(**************************************************************************************************************)
(*----------   P1 - ERECTOR   ----------*)
(* All P1 control bits and words must be within address MD3040~MD3079*)
(* All bits and words within the address will be reset when not in autorun mode*)
(**************************************************************************************************************)

	A1_RunStep 				AT %MW3040:INT;

(**************************************************************************************************************)
(*---------- P2 - EXIT ----------*)
(* All P2 control bits and words must be within address MD3080~MD3119*)
(* All bits and words within the address will be reset when not in autorun mode*)
(**************************************************************************************************************)
	A2_RunStep 				AT %MW3080:INT;

(**************************************************************************************************************)
(*---------- P3 - ELEVATOR ----------*)
(* All P3 control bits and words must be within address MD3120~MD3159*)
(* All bits and words within the address will be reset when not in autorun mode*)
(**************************************************************************************************************)

	A3_RunStep 				AT %MW3120		:INT;
	TapeReel_ActivatedL		AT %MX3122.0	:BOOL;
	TapeReel_ActivatedR		AT %MX3122.1	:BOOL;	
	
(**************************************************************************************************************)
(*---------- P4 - HORIZONTAL ----------*)
(* All P4 control bits and words must be within address MD3160~MD3199*)
(* All bits and words within the address will be reset when not in autorun mode*)
(**************************************************************************************************************)

	A4_RunStep 				AT %MW3160 :INT;

(**************************************************************************************************************)
(*---------- P5 SPARE ---------*)
(* All P5 control bits and words must be within address MD3200~MD3239*)
(* All bits and words within the address will be reset when not in autorun mode*)
(**************************************************************************************************************)

	A5_RunStep 				AT %MW3200:INT;

(**************************************************************************************************************)
(*---------- P6 SPARE ----------*)
(* All P6 control bits and words must be within address MD3240~MD3279*)
(* All bits and words within the address will be reset when not in autorun mode*)
(**************************************************************************************************************)

	A6_RunStep  			AT %MW3240 :INT;

(**************************************************************************************************************)
(*---------- P7 SPARE ----------*)
(* All P7 control bits and words must be within address MD3280~MD3319*)
(* All bits and words within the address will be reset when not in autorun mode*)
(**************************************************************************************************************)

	A7_RunStep 				AT %MW3280:INT;

(**************************************************************************************************************)
(*---------- P8 SPARE ----------*)
(* All P8 control bits and words must be within address MD3320~MD3359*)
(* All bits and words within the address will be reset when not in autorun mode*)
(**************************************************************************************************************)

	A8_RunStep 				AT %MW3320:INT;

	
	
	INPUT_TEST		AT %I* 	:INT;
	OUTPUT_TEST		AT %Q* 	:INT;

	I_Reset_HMI: BOOL;
END_VAR

// ---- GVLs/MC/GVL_Holding.TcGVL
VAR_GLOBAL RETAIN PERSISTENT
	
	(* Process Memory*)
	H_CO_StkRdyForXPush					:BOOL;	(*Stack Ready for X Pusher. Do not Stack up if ON*)
	H_CO_StkRdyForYPush					:BOOL;	(*Stack Ready for Y Pusher. Do not activate X Pusher if ON*)
	
	H_ServiceStop_Pressed				:BOOL;	(* Service Stop Pressed *)
	StackerFault_Triggered				:BOOL;
	XPusherFault_Triggered				:BOOL;
	YPusherFault_Triggered				:BOOL;
	ErectorFault_Triggered				:BOOL;
	ExitFault_Triggered					:BOOL;
	HorizontalFault_Triggered			:BOOL;
	MajorFault_Triggered				:BOOL;

		
	H_ER_CtnErected						:BOOL;	(*Carton Erected *)
	H_ER_CtnRdyForPushIn				:BOOL;	(*Carton Erected and Moving Side Flaps Closed. Ready for Stack Push In*)
	H_ER_CtnPushInDone					:BOOL;	(*Stack Pushed into Carton Done, Wait for Side Flap Close. Do not activate Push in if ON*)
	H_ER_CtnSideFlapDone				:BOOL;	(*Carton Side Flap Closing Done. Ready for Glueing*)
	H_ER_CtnRdyForGlue					:BOOL;	(*Carton Pushed into Exit Area Ready for Glueing.*)
	H_ER_CtnGlueDone					:BOOL;	(*Carton Glueing Done. Ready for Exit Send Out*)
	H_ER_CtnWeightOK					:BOOL;	(*Carton Weight Checking OK - At Glueing Area*)

	H_EL_CtnTapeDone					:BOOL;	(*Carton Tape Sealing Done - If ON, send out to exit during origin*)	
	H_EL_CtnWeightOK					:BOOL;	(*Carton Weight Checking OK - On Elevator*)
	H_CartonWeight						:REAL;
	
	H_HOR_CtnTapeDone					:BOOL;	(*Carton Tape Sealing Done - If ON, send out to exit during origin*)	
	H_HOR_CtnWeightOK					:BOOL;	(*Carton Weight Checking OK - On Elevator*)
	
	CaseBufferEmptying_Counter			:INT;
	CaseBufferEmptying_Setting			:INT;
	GlueEmptying_Counter				:INT;
	GlueEmptying_Setting				:INT;
	TapeLow_Setting						:INT;

	
	H_ER_WA_Srv_ZeroOffset				:REAL;	(*Set Zero Point for Case Min C = 180mm	*)
	H_ER_BufCvL_WA_Srv_ZeroOffset		:REAL;	(*Set Zero Point for Case Min B+C = 330mm, where B=2xFlap Width	*)
	H_ER_FlapL_WA_Srv_ZeroOffset		:REAL;	(*Set Zero Point for Case Min A = 200mm	*)
	H_ER_BufCvR_WA_Srv_ZeroOffset		:REAL;	(*Set Zero Point for Case Min B+C = 330mm, where B=2xFlap Width	*)
	H_ER_FlapR_WA_Srv_ZeroOffset		:REAL;	(*Set Zero Point for Case Min A = 200mm	*)
	H_EX_HeightL_WA_Srv_ZeroOffset		:REAL;	(*set Zero Point for Case Min B = 150mm*)
	H_EX_HeightR_WA_Srv_ZeroOffset		:REAL;	(*set Zero Point for Case Min B = 150mm*)
	H_EX_WA_Srv_ZeroOffset				:REAL;	(*Set Zero Point for Case Min C = 180mm*)
	H_CO_CV_WA_Srv_ZeroOffset			:REAL;	
	H_CO_Stopper_WA_Srv_ZeroOffset		:REAL;	
	H_EX_TopL_WA_Srv_ZeroOffset			:REAL;
	H_EX_TopR_WA_Srv_ZeroOffset			:REAL;
	H_CO_FFlapGuide_WA_Srv_ZeroOffset	:REAL;	(*Set Zero Point where Carton min A = 200mm*)

	H_CO_XPush_Srv_EndDatumPos:REAL;		(*Teach End Datum Point at Final Pushing Position for Carton min A = 200mm*)

	H_CO_YPush_Srv_BufFinalPos:REAL;		(*Teach Final Pushing Position to Push Stack onto Buffer Area Before Carton*)
	H_CO_YPush_Srv_CtnFinalPos:REAL;		(*Teach Final Pushing Position to Push Stack into Carton*)	
	H_CO_YPush_Srv_SafePosition:Real;	
	
	H_ER_Arm_Srv_CtnVacuumPos: REAL;		(*Teach Position for Erector cylinder to move up and ready for Vacuum*)
	H_ER_Arm_Srv_CtnErectPos: REAL;			(*Teach Position for Erector Arm to move to final carton erecting position*)

	H_EL_Srv_CtnLoadPos:REAL;				(*Teach Position for Elevator Carton Loading from Tilt Position*)
	H_EL_Srv_CtnRejectExitPos:REAL;			(*Teach Position for Elevator Reject Carton Exit Conveyor Position*)
	H_EL_Srv_CtnGoodExitPos:REAL;			(*Teach Position for Elevator Good Carton Exit Conveyor Position*)
	H_EL_Srv_TapeStartPos:REAL;				(*Teach Position for Elevator Taping Start Position (bottom)*)
	H_EL_Srv_TapeEndPos:REAL;				(*Teach Position for Elevator Taping End Position (Top)*)
 
	H_EL_Push_Srv_HomePos:REAL;				(*Set at Zero Point before Carton is pushed but need to avoid taping unit*)
	H_EL_Push_Srv_ExitfinalPos:REAL;		(*Teach Final Pushing Position to Push Carton onto Exit conveyors*)

	H_EL_Center_Srv_HomePos:REAL;			(*Set at Zero Point before to avoid Carton during tilting*)
	H_EL_Center_Srv_EndDatumPos:REAL;		(*Teach Position for Carton Centering to Tilt Vacuum ON for Carton min B=150mm*)
	H_EL_Center_Srv_MidDatumPos:REAL;		(*Teach Position for Elevator Carton Centering for Taping for Carton min B=150mm*)
	
	
	H_ER_Arm_Srv_HomePos: REAL;			
	H_CO_XPush_Srv_HomePos:REAL;			(*Set at Zero Point out of Bundle Stack Area*)
	H_CO_YPush_Srv_HomePos:REAL;			(*Set at Zero Point out of Bundle Buffer Area*)

	H_CO_XPush_Srv_CurrStandbyPos:REAL;			(* Calculated based on bundle size*)
	H_CO_YPush_Srv_CurrStandbyPos:REAL;			(* Calculated based on bundle size*)
	
	H_ER_WA_Srv_TargetPos				:REAL;
	H_ER_BufCvL_WA_Srv_TargetPos		:REAL;
	H_ER_FlapL_WA_Srv_TargetPos			:REAL;
	H_ER_BufCvR_WA_Srv_TargetPos		:REAL;
	H_ER_FlapR_WA_Srv_TargetPos			:REAL;
	H_EX_HeightL_WA_Srv_TargetPos		:REAL;
	H_EX_HeightR_WA_Srv_TargetPos		:REAL;
	H_EX_WA_Srv_TargetPos				:REAL;
	H_CO_CV_WA_Srv_TargetPos			:REAL;	
	H_CO_Stopper_WA_Srv_TargetPos		:REAL;
	H_EX_TopL_WA_Srv_TargetPos			:REAL;
	H_EX_TopR_WA_Srv_TargetPos			:REAL;
	H_CO_FFlapGuide_WA_Srv_TargetPos	:REAL;
	
	H_ER_ValveOffset					:REAL;	
	H_ER_1St_GlueStartPos				:REAL;
	H_ER_1St_GlueStopPos				:REAL;	
	H_ER_2nd_GlueStartPos				:REAL;
	H_ER_2nd_GlueStopPos				:REAL;		
	ER_GlueHold_Time					:TIME;
	
	
	H_CO_Bdl_StkX_Count:INT;	(*Current Stack X Count*)
	H_CO_Bdl_StkY_Count:INT;	(*Current Stack Y Count*)
	H_CO_Bdl_StkZ_Count:INT;	(*Current Stack Z Count*)

	H_CO_Bdl_StkX_Full:BOOL;	(*Current Stack X Full*)
	H_CO_Bdl_StkY_Full:BOOL;	(*Current Stack Y Full*)
	H_CO_Bdl_StkZ_Full:BOOL;	(*Current Stack Z Full*)
	
	
	
	(***************************** Statistic Value ******************************************)
	Statistic_Total_Runtime				:DINT;
	Statistic_Total_UpTime				:DINT;
	Statistic_Total_DownTime			:DINT;
	Statistic_Total_CaseProduce			:DINT;
	Statistic_Total_Good				:DINT;
	Statistic_Total_NG					:DINT;					
	
	Statistic_Man_Total_Runtime			:DINT;
	Statistic_Man_Total_UpTime			:DINT;
	Statistic_Man_Total_DownTime		:DINT;
	Statistic_Man_Total_CaseProduce		:DINT;
	Statistic_Man_Total_Good			:DINT;
	Statistic_Man_Total_NG				:DINT;
	
	Statistic_Shift_StartTimeH			:ARRAY [0..3] OF UINT;
	Statistic_Shift_StartTimeM			:ARRAY [0..3] OF UINT;
	Statistic_Shift_EndTimeH			:ARRAY [0..3] OF UINT;
	Statistic_Shift_EndTimeM			:ARRAY [0..3] OF UINT;	
	
	Statistic_PreviousShift_Number		:UINT;	
	Statistic_CurShift_Number			:UINT;	
	Statistic_CurShift_StartTime		:STRING;
	Statistic_CurShift_EndTime			:STRING;
	Statistic_CurShift_StartDate		:STRING;
	Statistic_CurShift_CaseProduce		:DINT;
	Statistic_CurShift_Good				:DINT;
	Statistic_CurShift_NG				:DINT;
	Statistic_CurShift_UpTime			:DINT;
	Statistic_CurShift_RunTime			:DINT;
	Statistic_CurShift_DownTime			:DINT;
	
	Statistic_Current					:structStatistic;
	Statistic_History					:structStatistic;
	Statistic_Manual					:structStatistic;
	Statistic_Total						:structStatistic;	
	
	Generate_Report						:BOOL;
	
(**************************************************************************************************************)
(* Exit Case Result *)
(**************************************************************************************************************)	
	Exit_Case_Good	:BOOL;
	Exit_Case_NG	:BOOL;	
END_VAR

// ---- GVLs/MC/GVL_Origin.TcGVL
{attribute 'Tc2GvlVarNames'}
VAR_GLOBAL

(**************************************************************************************************************)
(*----------   P0 - COLLATOR   ----------*)
(* All P0 control bits and words must be within address MD4000~MD4039*)
(* All bits and words within the address will be reset when not in autorun mode*)
(**************************************************************************************************************)

	AO0_RunStep					AT %MW4000:INT;

(**************************************************************************************************************)
(*----------   P1 - ERECTOR   ----------*)
(* All P1 control bits and words must be within address MD4040~MD4079*)
(* All bits and words within the address will be reset when not in autorun mode*)
(**************************************************************************************************************)

	AO1_RunStep 				AT %MW4040:INT;
	
(**************************************************************************************************************)
(*---------- P2 - EXIT ----------*)
(* All P2 control bits and words must be within address MD4080~MD4119*)
(* All bits and words within the address will be reset when not in autorun mode*)
(**************************************************************************************************************)
	AO2_RunStep 			AT %MW4080:INT;

(**************************************************************************************************************)
(*---------- P3 - ELEVATOR ----------*)
(* All P3 control bits and words must be within address MD4120~MD4159*)
(* All bits and words within the address will be reset when not in autorun mode*)
(**************************************************************************************************************)

	AO3_RunStep 			AT %MW4120:INT;

(**************************************************************************************************************)
(*---------- P4 HORIZONTAL----------*)
(* All P4 control bits and words must be within address MD4160~MD4199*)
(* All bits and words within the address will be reset when not in autorun mode*)
(**************************************************************************************************************)

	AO4_RunStep 			AT %MW4160 :INT;

(**************************************************************************************************************)
(*---------- P5 SPARE----------*)
(* All P5 control bits and words must be within address MD4200~MD4239*)
(* All bits and words within the address will be reset when not in autorun mode*)
(**************************************************************************************************************)

	AO5_RunStep 			AT %MW4200:INT;

(**************************************************************************************************************)
(*---------- P6 SPARE----------*)
(* All P6 control bits and words must be within address MD4240~MD4279*)
(* All bits and words within the address will be reset when not in autorun mode*)
(**************************************************************************************************************)

	AO6_RunStep  			AT %MW4240 :INT;

(**************************************************************************************************************)
(*---------- P7 SPARE----------*)
(* All P7 control bits and words must be within address MD4280~MD4319*)
(* All bits and words within the address will be reset when not in autorun mode*)
(**************************************************************************************************************)

	AO7_RunStep 			AT %MW4280:INT;

(**************************************************************************************************************)
(*---------- P8 SPARE ----------*)
(* All P8 control bits and words must be within address MD4320~MD4359*)
(* All bits and words within the address will be reset when not in autorun mode*)
(**************************************************************************************************************)

	AO8_RunStep 			AT %MW4320:INT;

	

END_VAR

// ---- GVLs/MC/GVL_Error.TcGVL
{attribute 'Tc2GvlVarNames'}
VAR_GLOBAL
	
(**************************************************************************************************************)
(* warning Flag *)
(**************************************************************************************************************)
W_ER_BufRefill		AT %MX2000.0:BOOL;
W_EX_TapeLRefill	AT %MX2000.1:BOOL;
W_EX_TapeRRefill	AT %MX2000.2:BOOL;
W_CO_IncomingEmpty	AT %MX2000.3:BOOL;
W_HOR_TapeLRefill	AT %MX2001.1:BOOL;
W_HOR_TapeRRefill	AT %MX2001.2:BOOL;
W_HOR_Conv_Full		AT %MX2001.3:BOOL;
W_Glue_Low_Level	AT %MX2001.4:BOOL;
W_Glue_is_Empty		AT %MX2001.5:BOOL;
W_CaseBuffer_is_Empty	AT %MX2001.6:BOOL;
W_ServiceStop		AT %MX2001.7:BOOL;
W_Hor_TapeLowL		AT %MX2002.0:BOOL;
W_Hor_TapeLowR		AT %MX2002.1:BOOL;

(**************************************************************************************************************)
(*General  Error Flag *)
(**************************************************************************************************************)

E_AutorunDataNG :STRING;
E_Erector_FrontDoor_Opn		:BOOL;
E_Erector_RearDoor_Opn		:BOOL;
E_Collator_FrontDoor_Opn	:BOOL;
E_Collator_RearDoor_Opn		:BOOL;
E_Elevator_LeftTopDoor_Opn	:BOOL;
E_Elevator_LeftBtmDoor_Opn	:BOOL;
E_Elevator_RightDoor_Opn	:BOOL;
E_Horizontal_LeftDoor_Opn	:BOOL;
E_Horizontal_RightDoor_Opn	:BOOL;
E_Door_SafetyBroken			:BOOL;
E_Estop_Panel				:BOOL;
E_Estop_Collator			:BOOL;
E_Estop_HorLeft				:BOOL;
E_Estop_HorRight			:BOOL;
E_Estop_HorExit				:BOOL;
E_EStop_SafetyBroken		:BOOL;
E_X_Axis_BundleStackCount	:BOOL;
E_Y_Axis_BundleStackCount	:BOOL;
E_Z_Axis_BundleStackCount	:BOOL;
E_Recipe_H_OutOfTolerance	:BOOL;
E_Recipe_L_OutOfTolerance	:BOOL;
E_Recipe_W_OutOfTolerance	:BOOL;
E_Recipe_A_OutOfTolerance	:BOOL;
E_Recipe_B_OutOfTolerance	:BOOL;
E_Recipe_C_OutOfTolerance	:BOOL;
E_Recipe_A_SmallerThan_W	:BOOL;
E_Recipe_C_SmallerThan_L	:BOOL;
E_Recipe_B_SmallerThan_H	:BOOL;
	
(**************************************************************************************************************)
(*P0  Error Flag *)
(* All P0 control bits and words must be within address MD1000~MD1039*)
(* All bits and words within the address will be reset when error reset*)
(**************************************************************************************************************)
	
	E_Stack_Overflow 						:BOOL;
	E_Stack_Full			AT %MX1000.1	:BOOL;
	E_Door_Open				AT %MX1000.2	:BOOL;
	E_Bundle_Stuck_on_Infeed AT %MX1000.3	:BOOL;
	E_Bundle_Full			AT %MX1000.4	:BOOL;
	E_CAM_Up_Timeout		AT %MX1000.5	:BOOL;
	E_BundleJam_AfterStack	AT %MX1000.6	:BOOL;
	E_BundleJam_atRelease	AT %MX1000.7	:BOOL;	
	E_CAM_Down_Timeout		AT %MX1001.0	:BOOL;
	E_Stack_Full_ON			AT %MX1001.1	:BOOL;
	E_BundleDetected		AT %MX1001.2	:BOOL;
	E_Bundle_Stack_Sensor	AT %MX1001.3	:BOOL;
	E_BundleDetect_Sensor1	AT %MX1002.0	:BOOL;
	E_BundleDetect_Sensor2	AT %MX1002.1	:BOOL;
	E_BundleDetect_Sensor3	AT %MX1002.2	:BOOL;
	E_BundleDetect_Sensor4	AT %MX1002.3	:BOOL;
	E_BundleDetect_Sensor5	AT %MX1002.4	:BOOL;
	E_BundleDetect_Sensor6	AT %MX1002.5	:BOOL;
	E_BundleDetect_Sensor7	AT %MX1002.6	:BOOL;
	E_BundleDetect_Sensor8	AT %MX1002.7	:BOOL;
	
	
(**************************************************************************************************************)
(*P1  Error Flag *)
(* All P1 control bits and words must be within address MD1040~MD1079*)
(* All bits and words within the address will be reset when error reset*)
(**************************************************************************************************************)

	E_Buff1_BundleNotDetect	AT %MX1040.0	:BOOL;
	E_BundleJam_atStaker	AT %MX1040.1	:BOOL;


(**************************************************************************************************************)
(*P2  Error Flag *)
(* All P2 control bits and words must be within address MD1080~MD1119*)
(* All bits and words within the address will be reset when error reset*)
(**************************************************************************************************************)

	E_Buf1_BundleMissing	AT %MX1080.0	:BOOL;	
	E_Buf1_BundleJam		AT %MX1080.1	:BOOL;
	E_GapSensor				AT %MX1080.2	:BOOL;
	E_BundleDetectedinBuf1	AT %MX1080.3	:BOOL;
	E_BundleDetectedinBuf2	AT %MX1080.4	:BOOL;
	E_GapSensorError		AT %MX1080.5	:BOOL;
	E_PTC_BundleNOK			AT %MX1080.6	:BOOL;
	E_Buf1_Sensor			AT %MX1080.7	:BOOL;
	E_Buf2_Sensor			AT %MX1081.0	:BOOL;
	
(**************************************************************************************************************)
(*P3  Error Flag *)
(* All P3 control bits and words must be within addres MD1120~MD1159*)
(* All bits and words within the address will be reset when error reset*)
(**************************************************************************************************************)

	E_NoGapAtStoper				AT %MX1120.0	:BOOL;	
	E_LeftStopper_NotDetect		AT %MX1120.1	:BOOL;	
	E_RightStopper_NotDetect 	AT %MX1120.2	:BOOL;		
	E_ER_BufRefill				AT %MX1120.3	:BOOL;
	E_CaseDetected				AT %MX1120.4	:BOOL;
	E_CaseNotDetected			AT %MX1120.5	:BOOL;
	E_CaseVacuumNotDetected		AT %MX1120.6	:BOOL;
	E_Nordson_Alarm				AT %MX1120.7	:BOOL;
	E_EmptyCaseDetected			AT %MX1121.0	:BOOL;
	E_CaseBufferAlignment_Err	AT %MX1121.1	:BOOL;
	E_CaseBuffer_Not_Ready		AT %MX1121.2	:BOOL;
	E_CaseBuffer_EmptySensors	AT %MX1121.3	:BOOL;
	E_Case_Infeed_Safety_NOk	AT %MX1121.4	:BOOL;
	E_ER_EmptyL_PE				AT %MX1121.5	:BOOL;
	E_ER_BufferL_PE				AT %MX1121.6	:BOOL;
	E_ER_EmptyR_PE				AT %MX1121.7	:BOOL;
	E_ER_BufferR_PE				AT %MX1122.0	:BOOL;
	
(**************************************************************************************************************)
(*P4  Error Flag *)
(* All P4 control bits and words must be within address MD1160~MD1199*)
(* All bits and words within the address will be reset when error reset*)
(**************************************************************************************************************)
	E_WT_Conv_Jam				AT %MX1160.0	:BOOL;	
	E_CartonMissing				AT %MX1160.1	:BOOL;
	E_EX_CartonDetected			AT %MX1160.2	:BOOL;

(**************************************************************************************************************)
(*P5  Error Flag *)
(* All P5 control bits and words must be within address MD1200~MD1239*)
(* All bits and words within the address will be reset when error reset*)
(**************************************************************************************************************)
	E_BeltTension_Right_NOK		AT %MX1200.0	:BOOL;
	E_BeltTension_Left_NOK		AT %MX1200.1	:BOOL;
	E_DriveBeltTension_NOK		AT %MX1200.2	:BOOL;
	E_Weight_CV_CartonNotDetect AT %MX1200.3	:BOOL;
	E_Weight_CV_CartonDetect	AT %MX1200.4	:BOOL;
	E_EL_CartonNotDetect		AT %MX1200.5	:BOOL;
	E_Weigh_ReadingErr			AT %MX1200.6	:BOOL;
	E_Weigh_ConsecutiveErr		AT %MX1200.7	:BOOL;

	E_CartonTapingErrL							:BOOL;
	E_CartonTapingErrR							:BOOL;
(**************************************************************************************************************)
(*P6  Error Flag *)
(* All P6 control bits and words must be within address MD1240~MD1279*)
(* All bits and words within the address will be reset when error reset*)
(**************************************************************************************************************)
	E_Top_Conv_Jam				AT %MX1240.0	:BOOL;
	E_Bottom_Conv_Jam			AT %MX1240.1	:BOOL;
	E_Hor_Entry_Sensor			AT %MX1240.2	:BOOL;
	E_Hor_Exit_Sensor			AT %MX1240.3	:BOOL;
	
(**************************************************************************************************************)
(*P7  Error Flag *)
(* All P7 control bits and words must be within address MD1280~MD1319*)
(* All bits and words within the address will be reset when error reset*)
(**************************************************************************************************************)

(**************************************************************************************************************)
(*P8  Error Flag *)
(* All P8 control bits and words must be within address MD1320~MD1359*)
(* All bits and words within the address will be reset when error reset*)
(**************************************************************************************************************)


END_VAR

// ---- GVLs/MC/GVL_Configuration.TcGVL
VAR_GLOBAL  RETAIN PERSISTENT
	A_Srv_XPusherHiSpeed	:REAL;
	A_Srv_XPusherLoSpeed	:REAL;
	A_Srv_YPusherHiSpeed	:REAL;
	A_Srv_YPusherLoSpeed	:REAL;	

	A_Srv_ErectorArmHiSpeed:REAL;
	A_Srv_ErectorArmLoSpeed:REAL;
	
	A_Srv_ElevAutoHiSpeed:REAL;
	A_Srv_ElevAutoLoSpeed:REAL;
	A_Srv_ElevAutoMidSpeed:REAL:=60000;
	
	
	A_Srv_BeltOriginSpeed:REAL:=10000;
	A_Srv_ElevOriginSpeed:REAL:=1000;
	A_Srv_WAOriginSpeed:REAL:=1000;
	
	A_Srv_BeltAutoHiSpeed:REAL:=50000;	(*200000*)
	A_Srv_BeltAutoLoSpeed:REAL:=30000;	

	A_Srv_Default_Acc:REAL:=1000;
	A_Srv_Default_Dec:REAL:=1000;

	(* 	1 = Operator
		2 = Maintenance
		3 = Supervisor
		4 = Flexlink 
	*)

	Cfg_UserLvl_Operation	:INT	:=1;		
	Cfg_UserLvl_Manual		:INT	:=2;
	Cfg_UserLvl_Recipe		:INT	:=3;
	Cfg_UserLvl_Setting		:INT	:=3;
	Cfg_UserLvl_Config		:INT	:=4;
	

	Cfg_EnbAutoWA			:BOOL	:=TRUE;		(*1=Enable Auto Width Adjust*)
	Cfg_VerticalExit		:BOOL	:=FALSE;	(*1=Enable Vertical Exit with elevator*)
	Cfg_CollDircLtoR		:BOOL	:=FALSE;		(*1=Collator Push In Direction from Left to Right, 0 = Right to Left*)
	Cfg_EnbNordson			:BOOL	:=FALSE;	(*1=Enable Nordson Glueing*)
	Cfg_EnbWeightCheck		:BOOL	:=TRUE;		(*1=Enable Weight Checking*)
	Cfg_HorizontalExit		:BOOL	:=TRUE;		(*1=Enable Horizontal Exit*)
	Cfg_Exit90DegConv		:BOOL	:= FALSE;	(* 1=Enable Exit 90 Deg Conveyor	*)
	Cfg_Upstream_Conveyor	:BOOL	:= TRUE;	(* Upstream conveyor is connected	*)
	Cfg_prodSpeed_perHour	:INT	:= 120;		(* Number of carton produce per minute *)
	
	
	Cfg_BypassCollator:BOOL	:= FALSE;	(*1=Bypass Collator to run Erector and Elevator only*)
	Cfg_BypassErector:BOOL	:= FALSE;	(*1=Bypass Erector to run Collator only*)
	Cfg_BypassHorizontal:BOOL:= FALSE;	(*1=Bypass Horizontal to run Collator only*)
	
	Cfg_CaseA_Min	:REAL	:= 200;	
	Cfg_CaseB_Min	:REAL	:= 150;	
	Cfg_CaseC_Min	:REAL	:= 180;	
	Cfg_BundleW_Min	:REAL	:= 20;	
	Cfg_BundleL_Min	:REAL	:= 70;	
	Cfg_BundleH_Min	:REAL	:= 15;

	Cfg_CaseA_Max	:REAL	:= 640;	
	Cfg_CaseB_Max	:REAL	:= 500;
	Cfg_CaseC_Max	:REAL	:= 640;	
	Cfg_BundleW_Max	:REAL	:= 300;	
	Cfg_BundleL_Max	:REAL	:= 320;	
	Cfg_BundleH_Max	:REAL	:= 150;	
	
END_VAR

// ---- GVLs/MC/GVL_HMI.TcGVL
VAR_GLOBAL
	
	NewRecipe:structRecipe;
	
	
	T_GlobalAckAlarm:BOOL;
	
	T_SimPushIn:BOOL;
	
	T_DisplayWordSelect:WORD;
	T_MonitorWord:WORD;
	T_MonitorByte1Name:STRING;
	T_MonitorByte2Name:STRING;
	T_Monitor2Bytes:BOOL;
	MC_WA_Run	:BOOL;
END_VAR

VAR_GLOBAL RETAIN PERSISTENT

	CurrRecipe		:structRecipe;
	McData			:structMachineData;
	HMI				:structHMI;
	T_GlueEnable	:BOOL;
	T_ExitCvFull	:BOOL;
	
END_VAR

// ---- GVLs/MC/GVL_Status.TcGVL
VAR_GLOBAL
	
END_VAR

// ---- GVLs/MC/GVL_Symbol_Spec.TcGVL
VAR_GLOBAL
	
(*FlexLink Standard Symbol Naming Convention*)
(*
ER = Erector
CO = Collator
EX = Exit
EL = Elevator
WT = Weight checker
PB = push button
PL = push button light
Emg = Emergency Stop
SC = Safety Circuit
Cyl = Cylinder
Srv = Servo Motor
Mtr = AC Motor
Nord = Nordson Dispenser
Alm = Alarm
Rdy = Ready
SFlapL = Side Flap Left
SFlapR = Side Flap Right
BFlapL = Bottom Flap Left
BFlapR = Bottom Flap Right
Stp = Stopper
Ctn = Carton
LC = Light Curtain
Bdl = Bundle
Stk = Stack
Push = Pusher
Brdg = Bridge
Fx = Fixed
Mv = Moving

SC[0] = COLLATOR STACKING
SC[1] = COLLATOR X PUSHER
SC[2] = COLLATOR Y PUSHER & BRIDGE
SC[3] = ERECTOR ARM & SIDE FLAP CLOSE
SC[4] = HOT GLUE & WEIGHT CHECKING 
SC[5] = TILT & ELEVATOR
SC[6] = HORIZONTAL

*)

END_VAR

// ---- GVLs/MC/GVL_Timer.TcGVL
VAR_GLOBAL
	
	CO_Stk_Up_TON: Ton;
	CO_Stk_Dn_TON: Ton;
	CO_Bdl_Count_TON: Ton;
	CO_Bdl_Reach_TON: Ton;
	CO_Bdl_Stack_TON: Ton;
	CO_Bdl_Count_TOFF: Ton;
	CO_Stk_AtBuf_TON: Ton;

	ER_BufCv_Ctn_TON:ton;
	ER_BufCvL_Ctn_TON:ton;
	ER_BufCvR_Ctn_TON:ton;

	TP_Cyl_Timeout: TIME := T#5S;
	
	EL_Ctn_TON: Ton;
	EL_Ctn_TOFF: Ton;
	EL_TopCv_Ctn_TON: Ton;
	EL_TopCv_Ctn_TOFF: Ton;
	EL_BotCv_Ctn_TON: Ton;
	EL_BotCv_Ctn_TOFF: Ton;
	
	CO_Bdl_ZFull_TON: Ton;
	CO_Bdl_XFull_TON: Ton;
	CO_Bdl_ZFull_TOFF: Ton;
	
	pls_CoStkMtrStop: R_trig;
	tmr_CoStkMtrStop: Ton;

	EL_LC_Safety_TON: Ton;
	
	HOR_Ctn_TON: Ton;
	HOR_Ctn_TOFF: Ton;
	HOR_DnStream_TOFF: Ton;
	HOR_TopCv_Ctn_TON: Ton;
	HOR_TopCv_Ctn_TOFF: Ton;
	HOR_BotCv_Ctn_TON: Ton;
	HOR_BotCv_Ctn_TOFF: Ton;
	
	HOR_LC_Safety_TON: Ton;
END_VAR

// ---- POUs/MC/MAIN.TcPOU
PROGRAM MAIN
VAR
	Reset: BOOL;
	MachineEmpty: BOOL;
	plsMemoryReset: R_trig;
	tmrStartWrite: Ton;
	tmrWriteInterval: Ton;
	WritePersistentDataBusy: BOOL;
	plsStartWrite: R_trig;
	InstWritePersistentData:WritePersistentData;
	Timeout:ton;
	Test: BOOL;
	TIMEr: TIME;
	plsPurgeErectorCaseOff	: 	R_trig;
	plsServiceStop			:	R_trig;
	plsMAchineStart			:	R_trig;
	WA_ResetDly:TON;
	MC_Empty:BOOL;
	GetUPSStatus:FB_GetUPSStatus;
	GetFB_LocalSystemTime:FB_LocalSystemTime;
END_VAR


(**************************************************************************************************************)
(* Machine Control *)
(**************************************************************************************************************)

HMI.V_MachineSpeed	:= 100;

Check_AutorunCond();

Check_Ethercat();

MC_Ctrl(
	In_Start_PB					:= I_Start_PB AND NOT W_ServiceStop AND ER_origin.ER_WA_Origin  ,
	In_Stop_PB					:= I_Stop_PB ,
	In_EmgOK					:= I_Emg_SC_OK AND NOT  E_EStop_SafetyBroken,
	In_Door_Sw					:= TRUE(*I_Door_SC_OK AND NOT E_Door_SafetyBroken*),
	In_Pressure_Sw				:= (I_PressSw_OK AND NOT I_Pneumatic_Sup1_ON AND NOT I_Pneumatic_Sup2_ON) OR NOT (I_Door_SC_OK AND Guard_door.Guard_Door_Fault) ,
	In_LightCurtainSafeToCross	:= TRUE(*HOR_LC_Muting*) ,
	In_LightCurtainOK			:= I_HLC_SC_OK  OR NOT I_Door_SC_OK OR Guard_door.Guard_Door_Fault,
	In_CommunicationOK			:= S_ECat_NOK,
	In_IncomingPowerPhase_OK	:= I_IncomingPowerPhase_OK,
	In_OtherTrouble				:= Guard_door.Guard_Door_Fault ,
	In_Reset_PB					:= I_Reset_PB OR I_Reset_HMI ,
	In_Start_Enable				:= A_AutorunDataOK ,
	In_EndProdWPCleared			:= ,
	In_WaitingForMaterial		:= NOT(I_Nord_Rdy OR NOT T_GlueEnable OR mc.DryRun) OR W_Glue_is_Empty	OR W_CaseBuffer_is_Empty,	
	Out_RedTower				=> O_Red_TL ,
	Out_YelTower				=> O_Yel_TL ,
	Out_GrnTower				=> O_Grn_TL ,
	Out_Buzzer					=> O_Buz_TL, 
	Out_StartPL					=> O_Start_PL,
	Out_StopPL					=> O_Stop_PL,
	Out_ResetPL					=> O_Reset_PL,
	McVar 						:= MC,	
	HMI 						:= HMI);


// ************************************************
// Service Stop Memory
IF I_Stop_PB AND mc.autorunning THEN 
	H_ServiceStop_Pressed	:= TRUE;
END_IF

plsMAchineStart	(CLK:= mc.AutoRunning);
IF plsMAchineStart.Q	THEN
	H_ServiceStop_Pressed	:= FALSE;
	MajorFault_Triggered 	:= FALSE;
	StackerFault_Triggered 	:= FALSE;
	XPusherFault_Triggered 	:= FALSE;
	YPusherFault_Triggered 	:= FALSE;
	ErectorFault_Triggered	:= FALSE;
	ExitFault_Triggered		:= FALSE;
	HorizontalFault_Triggered:= FALSE;
END_IF

// *************************************************	
// Service Stop Warning
plsServiceStop (CLK := H_ServiceStop_Pressed AND NOT mc.AutoRunning );
IF plsServiceStop.Q THEN
	W_ServiceStop	:= TRUE;	
END_IF	



// Machine Empty	
MachineEmpty := NOT I_ER_StpL_Ctn_PE AND
				NOT I_ER_StpR_Ctn_PE AND
				NOT I_EX_Cv_Ctn_PE AND
				NOT I_HOR_Entry_Cv_Present AND
				MC.AllStationRdy;

				
O_DoorLock	:= 	(* MC.ManualMode AND 
				I_Pneumatic_Sup1_ON AND 
				I_Pneumatic_Sup2_ON AND*)
				NOT (	mc.AutoRunning OR 
						SC[0].OriginSchRun OR
						SC[1].OriginSchRun OR
						SC[2].OriginSchRun OR
						SC[3].OriginSchRun OR
						SC[4].OriginSchRun OR
						SC[5].OriginSchRun OR
						SC[6].OriginSchRun);				

				
IF 	HMI.T_EndProd AND 
	sc[0].Rdy AND
	sc[1].Rdy AND
	sc[2].Rdy AND
	sc[3].Rdy AND
	sc[4].Rdy AND
	sc[6].Rdy AND	
	MachineEmpty AND
 	mc.AutoRunning THEN
	MC.StopPressed	:= TRUE;
END_IF


IF NOT mc.AutoRunning THEN
	HMI.T_EndProd := FALSE;
END_IF

(**************************************************************************************************************)
(* Calling of Programs *)
(**************************************************************************************************************)
WarningMsg();
Calc_McPerformance();
Std_System_Out();
TouchScreen();
Statistic();
Recipe_Handling();
Guard_Door();
Emergency_Stop();
CO_Main();			(*COLLATOR MAIN PROGRAM*)
ER_Main();			(*ERECTOR MAIN PROGRAM*)
EX_Main();			(*EXIT MAIN PROGRAM*)
(*EL_Main();		(*ELEVATOR MAIN PROGRAM*)*)
HMI.T_Station_BypassP[5] := TRUE;
HOR_Main();			(*HORIZONTAL MAIN PROGRAM*)
Track_and_Trace(); 	(* TRACK AND TRACE PROGRAM *)


(* MACHINE CONDITION *)
MC_Empty	:= NOT( 	I_CO_YStk_AtBuf1_PE OR 
						I_CO_YStk_AtBuf2_PE OR
						I_CO_Bdl_Stack_PE OR
						I_CO_Bdl_PE1 OR
						I_CO_Bdl_PE2 OR
						I_CO_Bdl_PE3 OR
						I_CO_Bdl_PE4 OR
						I_CO_Bdl_PE5 OR
						I_CO_Bdl_ZLimit_PE OR
						I_CO_Bdl_ZFull_PE OR
						I_ER_RefillL_PE OR
						I_ER_BufferL_PE OR
						I_ER_BufferR_PE OR
						I_ER_StpL_Ctn_PE OR
						I_ER_StpR_Ctn_PE OR
						I_EX_Cv_Ctn_PE OR
						I_HOR_Entry_Cv_Present									
												);


IF NOT MC.AutoMode THEN
	Memory_Handling();
END_IF

WA_ResetDly	(IN := NOT (sc[0].OriginSchRun OR
		sc[1].OriginSchRun OR
	 	sc[2].OriginSchRun OR 
		sc[3].OriginSchRun OR
		sc[4].OriginSchRun OR 
		sc[6].OriginSchRun OR	
		HMI.T_OriginSearch OR
		MC.OriginSchRun) AND 
		MC.AllOrigin AND
		MC_WA_Run , pt := T#1S);

		
IF WA_ResetDly.Q THEN
	MC_WA_Run	:=FALSE;
END_IF			

(**************************************************************************************************************)
(* UPS Battery Status *)
(**************************************************************************************************************)
GetUPSStatus(
	sNetId:= '10.1.33.138.1.1' , 
	nPort:= 801, 
	bEnable:=TRUE , 
	bValid=> , 
	bError=> , 
	nErrId=> , 
	stStatus=> );

END_PROGRAM

// ---- POUs/MC/Check_AutorunCond.TcPOU
PROGRAM Check_AutorunCond
VAR
END_VAR


E_AutorunDataNG := '';

	
IF (CurrRecipe.rCaseA < Cfg_CaseA_Min) OR 
	(CurrRecipe.rCaseA > Cfg_CaseA_Max) THEN
	E_AutorunDataNG := 'Case Dimension A out of tolerance';
	E_Recipe_A_OutOfTolerance	:= TRUE;
ELSE
	E_Recipe_A_OutOfTolerance	:= FALSE;
END_IF
	
IF (CurrRecipe.rCaseB < Cfg_CaseB_Min) OR 
	(CurrRecipe.rCaseB > Cfg_CaseB_Max) THEN
	E_AutorunDataNG := 'Case Dimension B out of tolerance';
	E_Recipe_B_OutOfTolerance	:= TRUE;
ELSE
	E_Recipe_B_OutOfTolerance	:= FALSE;
END_IF
	
IF (CurrRecipe.rCaseC < Cfg_CaseC_Min) OR 
	(CurrRecipe.rCaseC > Cfg_CaseC_Max) THEN
	E_AutorunDataNG := 'Case Dimension C out of tolerance';
	E_Recipe_C_OutOfTolerance	:= TRUE;
ELSE
	E_Recipe_C_OutOfTolerance	:= FALSE;
END_IF
		

IF 	E_Recipe_A_OutOfTolerance	OR
	E_Recipe_B_OutOfTolerance	OR
	E_Recipe_C_OutOfTolerance	
THEN	
	A_AutorunDataOK := FALSE;
ELSE
	A_AutorunDataOK := TRUE;	
END_IF

END_PROGRAM

// ---- POUs/MC/Check_Ethercat.TcPOU
PROGRAM Check_Ethercat
VAR
END_VAR


S_ECat_NOK := FALSE;


IF NOT ER.Bypass THEN
	S_ECat_NOK := 	 S_ECat_NOK 
					 OR (I_ECat_41BC1<>8)
					 OR (I_ECat_41DI1<>8)
					 OR (I_ECat_41DI2<>8)
					 OR (I_ECat_41DO1<>8)
					 OR (I_ECat_41DO2<>8)
					(* OR (I_ECat_41CO1<>8)	*)
					 OR (I_ECat_41BC2<>8)
					 OR (I_ECat_41BC3<>8)
					 OR (I_ECat_70A1<>8)
					 OR (I_ECat_71A1<>8)
					 OR (I_ECat_60A1<>8)
					 OR (I_ECat_61A1<>8)
					 OR (I_ECat_62A1<>8)
					 OR (I_ECat_63A1<>8)
					 OR (I_ECat_64A1<>8)
					 OR (I_ECat_65A1<>8)
					 OR (I_ECat_66A1<>8);
END_IF


IF NOT CO.Bypass THEN
	S_ECat_NOK := 		S_ECat_NOK 
					OR (I_ECat_141BC1<>8)
					OR (I_ECat_141DI1<>8)
					OR (I_ECat_141DO1<>8)
					OR (I_ECat_141BC2<>8)
					OR (I_ECat_170A1<>8) 
					OR (I_ECat_160A1<>8)
					OR (I_ECat_161A1<>8)
					OR (I_ECat_162A1<>8)
					OR (I_ECat_162A1<>8);
END_IF



IF NOT HOR.Bypass THEN
	S_ECat_NOK := S_ECat_NOK (*
					OR (I_ECat_241BC1<>8)
					OR (I_ECat_241DI1<>8)
					OR (I_ECat_241DO1<>8)*)
					OR (I_ECat_260A1<>8);
END_IF

END_PROGRAM

// ---- POUs/Erector/ER_Origin.TcPOU
PROGRAM ER_Origin
VAR_IN_OUT
	Station		:structStationCtrl;
END_VAR
VAR
	pls_OriginSchRun: R_trig;
	ER_CtnPresent_Origin:BOOL;
	ER_NoCtnPresent_Origin:BOOL;
	
	ER_WA_Origin: BOOL;
	ER_CtnDone_Origin: BOOL;
	ER_Ctn_OriginState: BOOL;
	TimeoutTrigger: BOOL;
	TimeoutSetting: TIME;
	Timeout:ton;
END_VAR

(**************************************************************************************************************)
(* Station Width Adjust in Origin Condition *)
(**************************************************************************************************************)
ER_WA_Origin := fcCompareWAPos(CurrPos:= ER_WA_Srv_Var.Out_CurrPos, TargetPos:= H_ER_WA_Srv_TargetPos) ;

(**************************************************************************************************************)
(* Station Origin Condition *)
(**************************************************************************************************************)

IF Cfg_CollDircLtoR THEN
	ER_CtnPresent_Origin := (	ER_StpR_Cyl_Var.S_WorkPos AND 
								ER_StpL_Cyl_Var.S_WorkPos AND
								ER_FFlapL_Cyl_Var.S_HomePos AND 
								(*ER_RFlapL_Cyl_Var.S_HomePos AND*)
								ER_FFlapR_Cyl_Var.S_HomePos AND 
								(*ER_RFlapR_Cyl_Var.S_WorkPos AND*)
								ER_TFlapClsL_Cyl_Var.S_WorkPos AND
								ER_TFlapClsR_Cyl_Var.S_WorkPos AND
							(*	ER_BFlapL_Vac_Var.S_Vacuum AND 
								ER_BFlapR_Vac_Var.S_Vacuum AND*)
								I_ER_StpL_Ctn_PE AND I_ER_StpR_Ctn_PE) 
								OR MC.DryRun ;
ELSE
	ER_CtnPresent_Origin := (	ER_StpR_Cyl_Var.S_WorkPos AND 
								ER_StpL_Cyl_Var.S_WorkPos AND
								ER_FFlapL_Cyl_Var.S_WorkPos AND 
								ER_RFlapL_Cyl_Var.S_WorkPos AND
								ER_FFlapR_Cyl_Var.S_HomePos AND 
								ER_RFlapR_Cyl_Var.S_HomePos AND
								(*
								ER_BFlapL_Vac_Var.S_Vacuum AND 
								ER_BFlapR_Vac_Var.S_Vacuum AND*)
								ER_BFlapCloseL_Cyl_Var.S_HomePos AND 
								ER_BFlapCloseR_Cyl_Var.S_HomePos AND
								I_ER_StpL_Ctn_PE AND I_ER_StpR_Ctn_PE)
								OR MC.DryRun ;
END_IF

ER_CtnDone_Origin := (	ER_StpR_Cyl_Var.S_WorkPos AND 
						ER_StpL_Cyl_Var.S_WorkPos AND
						ER_FFlapL_Cyl_Var.S_HomePos AND 
						ER_RFlapL_Cyl_Var.S_WorkPos AND
						ER_FFlapR_Cyl_Var.S_HomePos AND 
						ER_RFlapR_Cyl_Var.S_WorkPos AND
					(*	ER_BFlapCloseL_Cyl_Var.S_WorkPos AND 
						ER_BFlapCloseR_Cyl_Var.S_WorkPos AND*)
						I_ER_StpL_Ctn_PE AND I_ER_StpR_Ctn_PE) 
						OR MC.DryRun ;


ER_NoCtnPresent_Origin := (	ER_StpR_Cyl_Var.S_HomePos AND 
							ER_StpL_Cyl_Var.S_HomePos AND
							ER_FFlapL_Cyl_Var.S_HomePos AND 
							ER_RFlapL_Cyl_Var.S_HomePos AND
							ER_FFlapR_Cyl_Var.S_HomePos AND 
							ER_RFlapR_Cyl_Var.S_HomePos AND
							ER_TFlapOpnL_Cyl_var.S_HomePos AND
							ER_TFlapClsL_Cyl_var.S_HomePos AND
							ER_TFlapOpnR_Cyl_var.S_HomePos AND
							ER_TFlapClsR_Cyl_var.S_HomePos AND
							ER_CaseGuideL_Cyl_Var.S_HomePos AND
							ER_CaseGuideR_Cyl_Var.S_HomePos AND
							NOT I_ER_StpL_Ctn_PE AND 
							NOT I_ER_StpR_Ctn_PE)
							OR MC.DryRun;

ER_Ctn_OriginState := 	((	H_ER_CtnRdyForPushIn OR H_ER_CtnPushInDone) OR 
							H_ER_CtnSideFlapDone AND 
							ER_CtnPresent_Origin) OR
							(	NOT H_ER_CtnRdyForPushIn AND 
								NOT H_ER_CtnPushInDone AND
						 		NOT H_ER_CtnSideFlapDone AND 
								ER_NoCtnPresent_Origin) OR
							(H_ER_CtnSideFlapDone AND ER_CtnDone_Origin);
							
Station.Origin 	:=	(	(ER_WA_Origin OR NOT MC_WA_Run )AND
						(	(ER_Arm_Vac_Var.S_Release AND
							 ER_ArmTilt_Cyl_Var.S_WorkPos) OR
							(ER_Arm_Vac_Var.S_Vacuum AND
							 ER_ArmTilt_Cyl_Var.S_HomePos) )	AND		
						ER_Ctn_OriginState AND
						ER_BFlapL_Cyl_Var.S_HomePos AND 
						ER_BFlapR_Cyl_Var.S_HomePos) AND	
						ER_Arm_Cyl_Var.S_HomePos AND 						
						(fcComparePos(CurrPos:= ER_Arm_Srv_Var.Out_CurrPos, TargetPos:= H_ER_Arm_Srv_CtnVacuumPos, Tolerance :=3 ) OR
						MC_WA_Run OR Erector_SafetySensorBypass) OR
						Station.Bypass;			
					 		
(**************************************************************************************************************)
(* Station Origin Step *)
(**************************************************************************************************************)

pls_OriginSchRun(CLK:= MC.OriginSchRun OR Station.OriginSchRun);
(*EL_EL_TapeLock_Var.In_OrgWork := ER_WA_Srv_Var.Out_Ready;*)

Timeout(IN:=TimeoutTrigger, PT:=TimeoutSetting);
IF Timeout.Q THEN
	TimeoutTrigger := FALSE;
END_IF

IF (MC.OriginSchRun OR Station.OriginSchRun) AND NOT Station.Bypass   THEN
	CASE Station.OriginRunStep OF

	0 : 	(************* Ready To Run ****************)
			IF NOT Station.Origin AND pls_OriginSchRun.Q THEN
				Station.OriginRunStep := Station.OriginRunStep+10;	
			END_IF

	10 : 	(************* Check Sensors Before Homing ****************)
			Station.Status 		:= 'Org10: Check Sensors Before Homing';
			Station.StatusInt	:= 120;
			
			IF (I_ER_StpL_Ctn_PE OR I_ER_StpR_Ctn_PE) AND  
				NOT (H_ER_CtnRdyForPushIn (*OR H_ER_CtnPushInDone OR H_ER_CtnSideFlapDone*)) THEN 	
				Station.SeqFaultWord 	:= 100;
				Station.SeqFaultString 	:= 'Origin: Carton on Erector is in undefined state. Remove Carton.';
				E_CaseDetected			:= TRUE;	
			ELSIF (I_ER_StpL_Ctn_PE AND NOT I_ER_StpR_Ctn_PE) THEN
				Station.SeqFaultWord 		:= 101;		
				Station.SeqFaultString 		:= 'Origin: Carton Not Detected at Right Stopper. Check Carton.';
				E_RightStopper_NotDetect	:= TRUE;		
			ELSIF (NOT I_ER_StpL_Ctn_PE AND I_ER_StpR_Ctn_PE) THEN
				Station.SeqFaultWord 		:= 102;					
				Station.SeqFaultString 		:= 'Origin: Carton Not Detected at Left Stopper. Check Carton.';
				E_LeftStopper_NotDetect		:= TRUE;	
			ELSIF NOT (I_ER_StpL_Ctn_PE AND I_ER_StpR_Ctn_PE) AND  
				(H_ER_CtnRdyForPushIn (* OR H_ER_CtnPushInDone OR H_ER_CtnSideFlapDone*)) THEN 	
				Station.SeqFaultWord 		:= 104;
				Station.SeqFaultString 		:= 'Origin: Carton Missing or Not Properly Erected. Check Carton.';
				E_CaseNotDetected			:= TRUE;
			ELSIF H_ER_CtnRdyForPushIn AND   
				NOT (ER_BFlapL_Vac_Var.S_Vacuum (*AND ER_BFlapR_Vac_Var.S_Vacuum*)) THEN
				Station.SeqFaultWord 		:= 103;	
				Station.SeqFaultString 		:= 'Origin: Empty Carton Not Held by Vacuum. Remove Carton';		
				H_ER_CtnRdyForPushIn 		:= FALSE;
				E_CaseVacuumNotDetected		:= TRUE;			 
			ELSE
				Station.OriginRunStep := Station.OriginRunStep+10;				
	    	END_IF


			
	20 : 	(************* Release Erector Arm Vacuum ****************)
			Station.Status 		:= 'Org20: Release Erector Arm Vacuum';
			Station.StatusInt	:= 258;
			
			ER_Arm_Vac_Var.In_OrgPurge := TRUE;
	
			IF ER_Arm_Vac_Var.S_Release THEN
				ER_Arm_Vac_Var.In_OrgPurge := FALSE;
				IF ((fcComparePos(CurrPos:= ER_Arm_Srv_Var.Out_CurrPos, TargetPos:= H_ER_Arm_Srv_CtnVacuumPos, Tolerance := 0.5)) AND
						ER_Arm_Srv_Var.Out_InPos AND ER_Arm_Srv_Var.Out_Ready) THEN
					Station.OriginRunStep := 40;	(*Tilt Cylinders does not need to move Down*)
				ELSE
					Station.OriginRunStep := Station.OriginRunStep+10;					
				END_IF
			END_IF 
	 			
	30 : 	(************* Erector Arm Cylinder Down and Tilt Bwd ****************)
			Station.Status 		:= 'Org30: Erector Arm Cylinder Down and Tilt Bwd';
			Station.StatusInt	:= 259;
			
			IF ER_Arm_Srv_Var.Out_CurrPos>= H_ER_Arm_Srv_CtnVacuumPos THEN

					Station.OriginRunStep := Station.OriginRunStep+10;	
			ELSE
				IF NOT (ER_Arm_Cyl_Var.S_WorkPos AND ER_ArmTilt_Cyl_Var.S_HomePos) THEN
					ER_Arm_Cyl_Var.In_OrgWork 		:= TRUE;
					ER_ArmTilt_Cyl_Var.In_OrgHome 	:= TRUE;
				ELSE
					ER_Arm_Cyl_Var.In_OrgWork 		:= FALSE;
					ER_ArmTilt_Cyl_Var.In_OrgHome 	:= FALSE;
					Station.OriginRunStep := Station.OriginRunStep+10;	
				END_IF 
			END_IF
			
	40 : 	(************* Erector Arm Servo Move to Home Pos and all cylinders Bwd ****************)
			Station.Status 		:= 'Org40: Erector Arm Move to Home and all cylinders Bwd ';
			Station.StatusInt	:= 260;
			
			ER_Arm_Srv_Var.In_PosCmd 			:= H_ER_Arm_Srv_CtnVacuumPos; 
			ER_Arm_Srv_Var.In_VelCmd 			:= A_Srv_ErectorArmLoSpeed;
			ER_Arm_Srv_Var.In_MoveAbs 			:= TRUE;
			
			IF NOT H_ER_CtnRdyForPushIn AND 		(*No Carton Origin Sequence*)
				NOT H_ER_CtnPushInDone AND
				NOT H_ER_CtnSideFlapDone THEN
				ER_FFlapR_Cyl_Var.In_OrgHome 	:= TRUE;
				ER_RFlapR_Cyl_Var.In_OrgHome 	:= TRUE;
				ER_FFlapL_Cyl_Var.In_OrgHome 	:= TRUE;
				ER_RFlapL_Cyl_Var.In_OrgHome 	:= TRUE;		
				ER_BFlapL_Vac_Var.In_OrgPurge 	:= TRUE;	
				(*ER_BFlapR_Vac_Var.In_OrgPurge 	:= TRUE;*)
				ER_StpR_Cyl_Var.In_OrgHome 		:= TRUE;
				ER_StpL_Cyl_Var.In_OrgHome 		:= TRUE;	
				ER_TFlapOpnL_Cyl_var.In_OrgHome	:= TRUE;
				ER_TFlapClsL_Cyl_var.In_OrgHome	:= TRUE;
				ER_TFlapOpnR_Cyl_var.In_OrgHome	:= TRUE;
				ER_TFlapClsR_Cyl_var.In_OrgHome	:= TRUE;
				ER_CaseGuideL_Cyl_Var.In_OrgHome:= TRUE;
				ER_CaseGuideR_Cyl_Var.In_OrgHome:= TRUE;
				
				
			ELSE
				IF (H_ER_CtnRdyForPushIn OR
				H_ER_CtnPushInDone) AND 		(*Empty or Full Carton Origin Sequence*)
				NOT H_ER_CtnSideFlapDone THEN
					ER_BFlapL_Vac_Var.In_OrgVacuum 		:= TRUE;	
					(*ER_BFlapR_Vac_Var.In_OrgVacuum 		:= TRUE;*)			
					ER_BFlapCloseL_Cyl_Var.In_OrgHome 	:= TRUE;
					ER_BFlapCloseR_Cyl_Var.In_OrgHome 	:= TRUE;
					ER_StpR_Cyl_Var.In_OrgWork 			:= TRUE;
					ER_StpL_Cyl_Var.In_OrgWork 			:= TRUE;
					IF ER_BFlapL_Cyl_Var.S_HomePos AND
						ER_BFlapR_Cyl_Var.S_HomePos THEN
						IF Cfg_CollDircLtoR THEN
							ER_FFlapR_Cyl_Var.In_OrgWork := TRUE;
							ER_RFlapR_Cyl_Var.In_OrgWork := TRUE;	
							ER_FFlapL_Cyl_Var.In_OrgHome := TRUE;
							ER_RFlapL_Cyl_Var.In_OrgHome := TRUE;		
						ELSE
							ER_FFlapL_Cyl_Var.In_OrgWork := TRUE;
							ER_RFlapL_Cyl_Var.In_OrgWork := TRUE;			
							ER_FFlapR_Cyl_Var.In_OrgHome := TRUE;
							ER_RFlapR_Cyl_Var.In_OrgHome := TRUE;
						END_IF						
					END_IF
				ELSE								(*Fully closed Carton Origin Sequence*)
					ER_StpR_Cyl_Var.In_OrgWork := TRUE;
					ER_StpL_Cyl_Var.In_OrgWork := TRUE;		
					ER_BFlapL_Vac_Var.In_OrgPurge := TRUE;	
					(*ER_BFlapR_Vac_Var.In_OrgPurge := TRUE;*)	
					IF ER_BFlapL_Cyl_Var.S_HomePos AND
						ER_BFlapR_Cyl_Var.S_HomePos THEN
						ER_FFlapR_Cyl_Var.In_OrgHome := TRUE;
						ER_FFlapL_Cyl_Var.In_OrgHome := TRUE;
						ER_RFlapR_Cyl_Var.In_OrgWork := TRUE;	
						ER_RFlapL_Cyl_Var.In_OrgWork := TRUE;							
					END_IF	
					IF ER_RFlapR_Cyl_Var.S_WorkPos AND
						ER_RFlapL_Cyl_Var.S_WorkPos THEN
						ER_BFlapCloseL_Cyl_Var.In_OrgWork := TRUE;
						ER_BFlapCloseR_Cyl_Var.In_OrgWork := TRUE;						
					END_IF
				END_IF	
			END_IF			

			ER_BFlapL_Cyl_Var.In_OrgHome := TRUE;
			ER_BFlapR_Cyl_Var.In_OrgHome := TRUE;
			
			IF 	ER_Ctn_OriginState AND
				ER_BFlapL_Cyl_Var.S_HomePos AND 
				ER_BFlapR_Cyl_Var.S_HomePos AND	
				(ER_RFlapL_Cyl_Var.S_HomePos OR (ER_RFlapL_Cyl_Var.In_OrgWork AND ER_RFlapL_Cyl_Var.S_WorkPos))AND 		
				((fcComparePos(CurrPos:= ER_Arm_Srv_Var.Out_CurrPos, TargetPos:= H_ER_Arm_Srv_CtnVacuumPos, Tolerance := 0.5) AND
				ER_Arm_Srv_Var.Out_InPos AND ER_Arm_Srv_Var.Out_Ready) OR
				MC_WA_Run) THEN
				ER_Arm_Srv_Var.In_MoveAbs 		:= FALSE;
				ER_StpR_Cyl_Var.In_OrgHome 		:= FALSE;
				ER_StpL_Cyl_Var.In_OrgHome 		:= FALSE;
				ER_FFlapR_Cyl_Var.In_OrgHome 	:= FALSE;
				ER_RFlapR_Cyl_Var.In_OrgHome 	:= FALSE;
				ER_FFlapL_Cyl_Var.In_OrgHome 	:= FALSE;
				ER_RFlapL_Cyl_Var.In_OrgHome 	:= FALSE;		
				ER_BFlapL_Vac_Var.In_OrgPurge 	:= FALSE;	
				(*ER_BFlapR_Vac_Var.In_OrgPurge 	:= FALSE;*)
				ER_FFlapR_Cyl_Var.In_OrgWork 	:= FALSE;
				ER_RFlapR_Cyl_Var.In_OrgWork 	:= FALSE;	
				ER_FFlapL_Cyl_Var.In_OrgWork 	:= FALSE;
				ER_RFlapL_Cyl_Var.In_OrgWork 	:= FALSE;			
				ER_BFlapL_Vac_Var.In_OrgVacuum 	:= FALSE;	
				(*ER_BFlapR_Vac_Var.In_OrgVacuum 	:= FALSE;*)				
				ER_BFlapL_Cyl_Var.In_OrgHome 	:= FALSE;
				ER_BFlapR_Cyl_Var.In_OrgHome 	:= FALSE;
				ER_TFlapOpnL_Cyl_var.In_OrgHome	:= FALSE;
				ER_TFlapClsL_Cyl_var.In_OrgHome	:= FALSE;
				ER_TFlapOpnR_Cyl_var.In_OrgHome	:= FALSE;
				ER_TFlapClsR_Cyl_var.In_OrgHome	:= FALSE;
				ER_CaseGuideL_Cyl_Var.In_OrgHome:= FALSE;
				ER_CaseGuideR_Cyl_Var.In_OrgHome:= FALSE;
				Station.OriginRunStep := Station.OriginRunStep+10;	
			END_IF

	50 : 	(************* Erector Arm Cylinder Up and Tilt Fwd ****************)
			Station.Status 		:= 'Org50: Erector Arm Cylinder Up ';
			Station.StatusInt	:= 261;
			
			IF NOT ER_Arm_Cyl_Var.S_HomePos  THEN
				ER_Arm_Cyl_Var.In_OrgHome 		:= TRUE;
				ER_Arm_Cyl_Var.In_OrgWork 		:= FALSE;
			ELSE
				ER_Arm_Cyl_Var.In_OrgHome 		:= FALSE;
				ER_Arm_Cyl_Var.In_OrgWork 		:= FALSE;
				Station.OriginRunStep := Station.OriginRunStep+10;	
			END_IF 
			
	60:		(************* and Tilt Fwd ****************)
			Station.Status 		:= 'Org60: Tilt Fwd ';
			Station.StatusInt	:= 261;
			
			IF NOT ER_ArmTilt_Cyl_Var.S_WorkPos THEN
				ER_ArmTilt_Cyl_Var.In_OrgWork 	:= TRUE;
				ER_ArmTilt_Cyl_Var.In_OrgHome 	:= FALSE;
			ELSE
				ER_ArmTilt_Cyl_Var.In_OrgWork 	:= FALSE;
				ER_ArmTilt_Cyl_Var.In_OrgHome 	:= FALSE;
				
				IF NOT MC_WA_Run THEN
					Station.OriginRunStep := 0;
				ELSE
					Station.OriginRunStep := 1000;	
				END_IF	
			END_IF 		
	
	1000 : 	(************* Check Sensor Before Width Adjust ****************)
			Station.Status := 'Conveyor Run and Check Sensor Before Width Adjust';
			
			TimeoutTrigger := TRUE;
			TimeoutSetting := T#5S;
			
			
			IF I_ER_StpL_Ctn_PE THEN
				Station.SeqFaultWord 	:= 150;	
				E_CaseDetected			:=TRUE;		
				Station.SeqFaultString 	:= 'Origin: Carton Detected on Erector Left Stopper. Remove Carton for Width Adjustment';						 			
			ELSIF I_ER_StpR_Ctn_PE THEN
				Station.SeqFaultWord 	:= 151;	
				E_CaseDetected			:=TRUE;	
				Station.SeqFaultString 	:= 'Origin: Carton Detected on Erector Right Stopper. Remove Carton for Width Adjustment';							 			
			ELSIF  I_ER_BufferL_PE THEN
				Station.SeqFaultWord 	:= 152;	
				E_EmptyCaseDetected		:= TRUE;
				Station.SeqFaultString 	:= 'Origin: Carton Detected on Left Buffer Conveyor. Remove Carton Buffer for Width Adjustment';							 			
			ELSIF  I_ER_BufferR_PE THEN
				Station.SeqFaultWord 	:= 153;	
				E_EmptyCaseDetected		:= TRUE;		
				Station.SeqFaultString 	:= 'Origin: Carton Detected on Right Buffer Conveyor. Remove Carton Buffer for Width Adjustment';					 			
			ELSIF I_ER_RefillL_PE THEN
				Station.SeqFaultWord 	:= 154;	
				E_EmptyCaseDetected		:= TRUE;		
				Station.SeqFaultString 	:= 'Origin: Carton Detected on Left Buffer Conveyor. Remove Carton Buffer for Width Adjustment';					 			
			ELSIF Timeout.Q THEN
				ER_BufCvL_Mtr_Var.In_OrgOn := FALSE;
				Station.OriginRunStep := Station.OriginRunStep+10;	
			END_IF
	
	1010 : 	(************* Move All Erector WA to the right width ****************)
			
				
			EL_EL_TapeLock_Var.In_OrgWork		:= FALSE;
			ER_WA_Srv_Var.In_PosCmd 			:= H_ER_WA_Srv_TargetPos;
			ER_WA_Srv_Var.In_VelCmd 			:= A_Srv_WAOriginSpeed;
			ER_WA_Srv_Var.In_MoveAbs 			:= TRUE;
			Station.Status := 'Move Erector WA to the proper width';
				
			IF ER_WA_Origin THEN
				ER_WA_Srv_Var.In_ServoOn 		:= FALSE;
				ER_WA_Srv_Var.In_MoveAbs 		:= FALSE;
				Station.OriginRunStep 			:= 0;
			END_IF
						
	END_CASE

ELSE

	TimeoutTrigger := FALSE;
	Station.OriginRunStep := 0;	
	
END_IF

END_PROGRAM

// ---- POUs/FB/fcCompareWAPos.TcPOU
FUNCTION fcCompareWAPos : BOOL
VAR_INPUT
	CurrPos:REAL;
	TargetPos:REAL;
END_VAR
VAR
END_VAR

IF CurrPos >= (TargetPos-1) AND
	CurrPos <= (TargetPos+1) THEN
	fcCompareWAPos := TRUE;
ELSE
	fcCompareWAPos := FALSE;
END_IF

END_FUNCTION

// ---- POUs/FB/fcComparePos.TcPOU
FUNCTION fcComparePos : BOOL
VAR_INPUT
	CurrPos		:REAL;
	TargetPos	:REAL;
	Tolerance	:REAL;
END_VAR
VAR
END_VAR

IF CurrPos >= 	(TargetPos	-	Tolerance) AND
	CurrPos <= 	(TargetPos	+	Tolerance) THEN
	fcComparePos := TRUE;
ELSE
	fcComparePos := FALSE;
END_IF

END_FUNCTION

// ---- POUs/MC/Guard_Door.TcPOU
PROGRAM Guard_Door
VAR
	Guard_Door_Fault	:	BOOL;
	tmrGuardDoor		:	TON;
END_VAR

(*
Guard_Door_Fault	:= 	E_Erector_FrontDoor_Opn	OR
						E_Erector_RearDoor_Opn	OR
						E_Collator_FrontDoor_Opn OR
						E_Collator_RearDoor_Opn OR
						E_Elevator_LeftTopDoor_Opn OR
						E_Elevator_LeftBtmDoor_Opn OR
						E_Elevator_RightDoor_Opn OR
						E_Horizontal_LeftDoor_Opn OR
						E_Horizontal_RightDoor_Opn ;*)

tmrGuardDoor (IN := (Guard_Door_Fault AND I_Door_SC_OK ) OR (NOT Guard_Door_Fault AND not I_Door_SC_OK ), pt:= T#1S);
(*
IF tmrGuardDoor.Q THEN
E_Door_SafetyBroken	:= TRUE;						
END_IF											
*)

IF mc.ResetPressed THEN
	E_Erector_FrontDoor_Opn		:= FALSE;
	E_Erector_RearDoor_Opn		:= FALSE;
	E_Collator_FrontDoor_Opn	:= FALSE;
	E_Collator_RearDoor_Opn		:= FALSE;
	E_Elevator_LeftTopDoor_Opn	:= FALSE;
	E_Elevator_LeftBtmDoor_Opn	:= FALSE;
	E_Elevator_RightDoor_Opn	:= FALSE;
	E_Horizontal_LeftDoor_Opn	:= FALSE;
	E_Horizontal_RightDoor_Opn	:= FALSE;
	E_Door_SafetyBroken			:= FALSE;
END_IF
(*
IF not I_Erector_Front_Door_Sen THEN
	E_Erector_FrontDoor_Opn	:= TRUE;
END_IF

IF NOT I_Erector_Rear_Door_Sen THEN
	E_Erector_RearDoor_Opn	:= TRUE;
END_IF

IF NOT I_COL_Front_Door_Sen THEN
	E_Collator_FrontDoor_Opn	:=TRUE;
END_IF

IF NOT I_COL_Rear_Door_Sen THEN
	E_Collator_RearDoor_Opn	:=TRUE;
END_IF

IF NOT I_HOR_Left_Door THEN
	E_Horizontal_LeftDoor_Opn	:=TRUE;
END_IF

IF NOT I_HOR_Right_Door THEN
	E_Horizontal_RightDoor_Opn	:=TRUE;
END_IF
*)

END_PROGRAM

// ---- POUs/MC/WarningMsg.TcPOU
PROGRAM WarningMsg
VAR
END_VAR

(*
IF MC.AutoMode OR MC.ManualMode THEN
	
	IF W_ER_BufRefill THEN
		HMI.T_StatusString 		:= 'Erector Carton Buffer Conveyor Almost Empty. Refill Carton.';
		HMI.T_StatusStringInt	:= 20;			
	ELSIF W_EX_TapeLRefill THEN
		HMI.T_StatusString 		:= 'Left Tape Almost Empty. Refill Tape.';
		HMI.T_StatusStringInt	:= 21;	
	ELSIF W_EX_TapeRRefill THEN
		HMI.T_StatusString 		:= 'Right Tape Almost Empty. Refill Tape.';
		HMI.T_StatusStringInt	:= 22;	
	ELSIF W_HOR_TapeLRefill THEN
		HMI.T_StatusString 		:= 'Left Tape Almost Empty. Refill Tape.';
		HMI.T_StatusStringInt	:= 23;	
	ELSIF W_HOR_TapeRRefill THEN
		HMI.T_StatusString 		:= 'Right Tape Almost Empty. Refill Tape.';
		HMI.T_StatusStringInt	:= 24;			
	END_IF
END_IF
*)

END_PROGRAM

// ---- POUs/MC/Calc_McPerformance.TcPOU
PROGRAM Calc_McPerformance
VAR
	plsResetCycleTime:r_trig;
	CycleTimeCalc:REAL;
	IdleTimeCalc:real;
	plsResetIdleTime: R_trig;
	CalcRunTime:fbCalculateTotalTime;
	CalcIdleTime:fbCalculateTotalTime;
	CalcMajorDownTime:fbCalculateTotalTime;
	CalcMinorDownTime:fbCalculateTotalTime;
END_VAR

(************************************************************)
(* Calculate Machine Output									*)
(************************************************************)

IF H_EL_CtnWeightOK AND EL.RunStep=1000 THEN
	McData.Cnt_TotalGood := McData.Cnt_TotalGood + 1;
	McData.TotalRunCycles := McData.TotalRunCycles + 1;
ELSIF NOT H_EL_CtnWeightOK AND EL.RunStep=1000 THEN
	McData.Cnt_TotalNG := McData.Cnt_TotalNG + 1;
	McData.TotalRunCycles := McData.TotalRunCycles + 1;
END_IF

McData.Cnt_TotalOutput := McData.Cnt_TotalGood + McData.Cnt_TotalNG;

IF McData.Cnt_TotalOutput > 0 THEN
	McData.Cnt_TotalYield := UDINT_TO_REAL(McData.Cnt_TotalGood/McData.Cnt_TotalOutput) * 100;
ELSE
	McData.Cnt_TotalYield := 0;
END_IF

IF HMI.T_ResetCounters THEN
	McData.Cnt_TotalGood := 0;
	McData.Cnt_TotalNG := 0;
END_IF

(************************************************************)
(* Calculate Machine Cycle Time								*)
(************************************************************)

plsResetCycleTime(CLK:= MC.AutoRunning AND NOT MC.IdleState);
plsResetIdleTime(CLK:= MC.AutoRunning AND MC.IdleState);

IF plsResetCycleTime.Q THEN
	McData.CycleTimeSec := CycleTimeCalc;
	CycleTimeCalc := 0;
ELSIF plsResetIdleTime.Q THEN
	McData.IdleTimeSec := IdleTimeCalc;
	IdleTimeCalc := 0;
END_IF

IF MC.AutoRunning AND Clock100msOnPls THEN
	IF MC.IdleState THEN
		IdleTimeCalc := IdleTimeCalc + 0.1;
	ELSE
		CycleTimeCalc := CycleTimeCalc + 0.1;		
	END_IF
END_IF

IF McData.CycleTimeSecAvg <> 0 THEN
	McData.CycleTimeSecAvg := (McData.CycleTimeSecAvg + McData.CycleTimeSec)/2;
ELSE
	McData.CycleTimeSecAvg := McData.CycleTimeSec;
END_IF

IF McData.IdleTimeSecAvg <> 0 THEN
	McData.IdleTimeSecAvg := (McData.IdleTimeSecAvg + McData.IdleTimeSec)/2;
ELSE
	McData.IdleTimeSecAvg := McData.IdleTimeSec;
END_IF

(************************************************************)
(* Calculate Machine Run Time								*)
(************************************************************)

IF Clock1sOnPls THEN
	
	CalcRunTime(
		In_EnableCount:= MC.AutoRunning, 
		TotalHour=> McData.TotalRuntimeHour, 
		TotalMin=> McData.TotalRuntimeMin, 
		TotalSec=> McData.TotalRuntimeSec);

	CalcIdleTime(
		In_EnableCount:= NOT (MC.Trouble OR MC.StationStopErr OR MC.AutoRunning), 
		In_ResetCount := HMI.T_ResetTotalTime,
		TotalHour=> McData.TotalIdletimeHour, 
		TotalMin=> McData.TotalIdletimeMin, 
		TotalSec=> McData.TotalIdletimeSec);

	CalcMajorDownTime(
		In_EnableCount:= MC.Trouble, 
		In_ResetCount := HMI.T_ResetTotalTime,
		TotalHour=> McData.TotalMajorDowntimeHour, 
		TotalMin=> McData.TotalMajorDowntimeMin, 
		TotalSec=> McData.TotalMajorDowntimeSec);

	CalcMinorDownTime(
		In_EnableCount:= MC.StationStopErr, 
		In_ResetCount := HMI.T_ResetTotalTime,
		TotalHour=> McData.TotalMinorDowntimeHour, 
		TotalMin=> McData.TotalMinorDowntimeMin, 
		TotalSec=> McData.TotalMinorDowntimeSec);
		
END_IF

IF HMI.T_ResetTotalTime THEN
	McData.CycleTimeSec := 0;
	McData.CycleTimeSecAvg := 0;
	McData.IdleTimeSec := 0;
	McData.IdleTimeSecAvg := 0;
	McData.MTBA := 0;
	McData.MTBF := 0;
END_IF

END_PROGRAM

// ---- POUs/FB/fbCalculateTotalTime.TcPOU
FUNCTION_BLOCK fbCalculateTotalTime
VAR_INPUT
	In_EnableCount:BOOL;
	In_ResetCount:BOOL;
END_VAR
VAR_OUTPUT
	TotalHour	:DWORD;
	TotalMin	:INT;
	TotalSec	:INT;
END_VAR
VAR
END_VAR


IF In_EnableCount THEN
	TotalSec := TotalSec + 1;
	IF TotalSec >= 60 THEN
		TotalMin := TotalMin + 1;
		TotalSec := 0;
		IF TotalMin >= 60 THEN
			TotalHour := TotalHour + 1;
			TotalMin := 0;
		END_IF
	END_IF
END_IF

IF In_ResetCount THEN
	TotalHour	:=0;
	TotalMin	:=0;
	TotalSec	:=0;
END_IF

END_FUNCTION_BLOCK

// ---- POUs/MC/Std_System_Out.TcPOU
PROGRAM Std_System_Out
VAR

	Clk50ms:TON;
	ClkOff50ms:TON;
	Clk100ms:TON;
	ClkOff100ms:TON;
	Clk500ms:TON;
	ClkOff500ms:TON;
	ClkOn1s:TON;
	ClkOff1s:TON;

	T50ms_RTRIG: R_TRIG;
	T100ms_RTRIG: R_TRIG;
	T500ms_RTRIG: R_TRIG;
	T1s_RTRIG: R_TRIG;

END_VAR

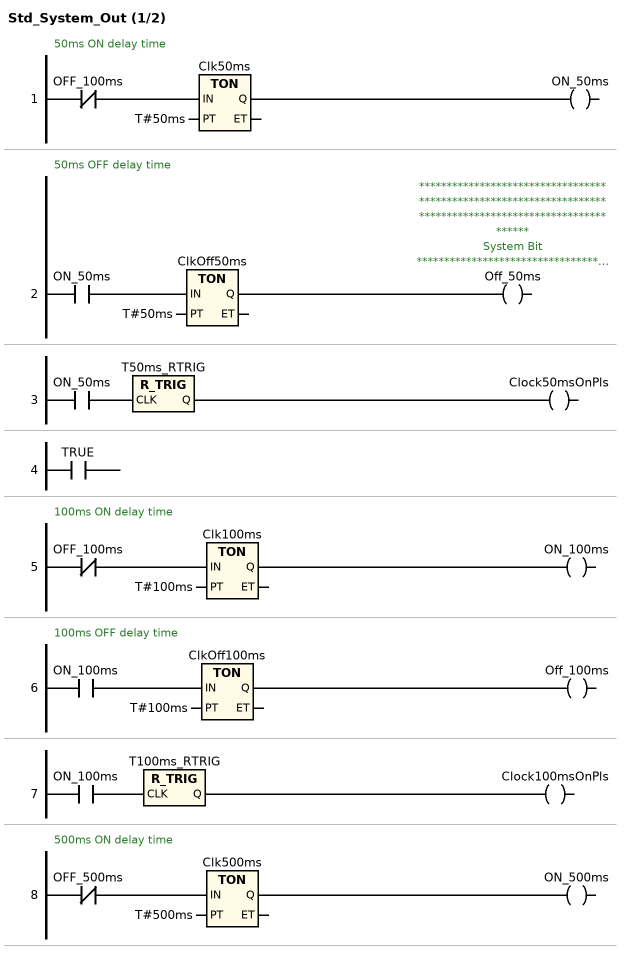
// NETWORK 1
// 50ms ON delay time
Clk50ms(IN := NOT OFF_100ms, PT := T#50ms); // TON
ON_50ms := Clk50ms.Q;

// NETWORK 2
// 50ms OFF delay time
//   Off_50ms: ************************************************************************************************************ System Bit ************************************************************************************************************
ClkOff50ms(IN := ON_50ms, PT := T#50ms); // TON
Off_50ms := ClkOff50ms.Q;

// NETWORK 3
T50ms_RTRIG(CLK := ON_50ms); // R_TRIG
Clock50msOnPls := T50ms_RTRIG.Q;

// NETWORK 4

// NETWORK 5
// 100ms ON delay time
Clk100ms(IN := NOT OFF_100ms, PT := T#100ms); // TON
ON_100ms := Clk100ms.Q;

// NETWORK 6
// 100ms OFF delay time
ClkOff100ms(IN := ON_100ms, PT := T#100ms); // TON
Off_100ms := ClkOff100ms.Q;

// NETWORK 7
T100ms_RTRIG(CLK := ON_100ms); // R_TRIG
Clock100msOnPls := T100ms_RTRIG.Q;

// NETWORK 8
// 500ms ON delay time
Clk500ms(IN := NOT OFF_500ms, PT := T#500ms); // TON
ON_500ms := Clk500ms.Q;

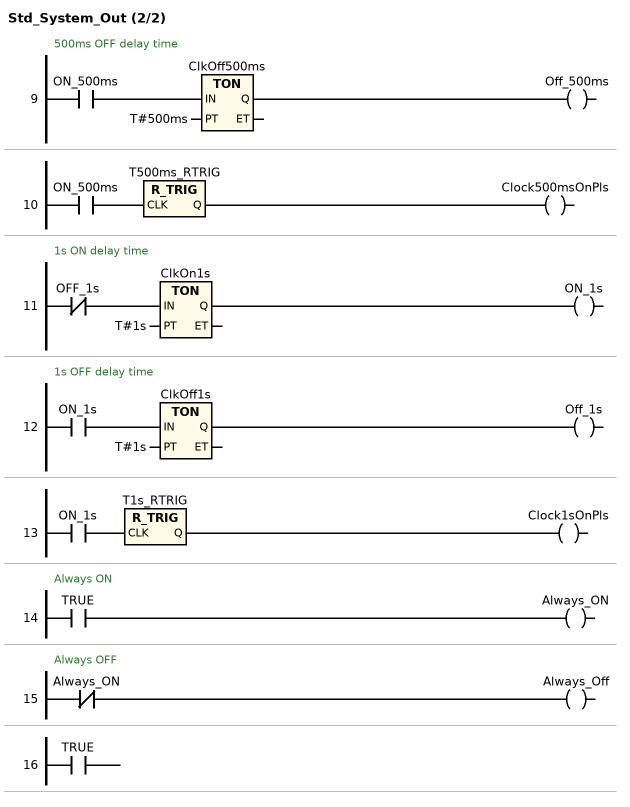
// NETWORK 9
// 500ms OFF delay time
ClkOff500ms(IN := ON_500ms, PT := T#500ms); // TON
Off_500ms := ClkOff500ms.Q;

// NETWORK 10
T500ms_RTRIG(CLK := ON_500ms); // R_TRIG
Clock500msOnPls := T500ms_RTRIG.Q;

// NETWORK 11
// 1s ON delay time
ClkOn1s(IN := NOT OFF_1s, PT := T#1s); // TON
ON_1s := ClkOn1s.Q;

// NETWORK 12
// 1s OFF delay time
ClkOff1s(IN := ON_1s, PT := T#1s); // TON
Off_1s := ClkOff1s.Q;

// NETWORK 13
T1s_RTRIG(CLK := ON_1s); // R_TRIG
Clock1sOnPls := T1s_RTRIG.Q;

// NETWORK 14
// Always ON
Always_ON := TRUE;

// NETWORK 15
// Always OFF
Always_Off := NOT Always_ON;

// NETWORK 16

END_PROGRAM

// ---- POUs/MC/TouchScreen.TcPOU
PROGRAM TouchScreen
VAR
END_VAR


CASE T_DisplayWordSelect OF

	0:
	T_MonitorWord  		:= IW_41DI1;
	T_MonitorByte1Name	:= 'IX0.x';
	T_MonitorByte2Name	:= 'IX1.x';
	T_Monitor2Bytes		:= TRUE;

	1:	
	T_MonitorWord  		:= IW_41DI2;
	T_MonitorByte1Name	:= 'IX2.x';
	T_MonitorByte2Name	:= 'IX3.x';
	T_Monitor2Bytes		:= TRUE;

	10:
	T_MonitorWord  		:= IW_60A1;
	T_MonitorByte1Name	:= 'IX10.x';
	T_MonitorByte2Name	:= '';
	T_Monitor2Bytes		:= FALSE;

	11:
	T_MonitorWord  		:= IW_61A1;
	T_MonitorByte1Name	:= 'IX11.x';
	T_MonitorByte2Name	:= '';
	T_Monitor2Bytes		:= FALSE;

	12:
	T_MonitorWord  		:= IW_62A1;
	T_MonitorByte1Name	:= 'IX12.x';
	T_MonitorByte2Name	:= '';
	T_Monitor2Bytes		:= FALSE;
	
	13:
	T_MonitorWord  		:= IW_63A1;
	T_MonitorByte1Name	:= 'IX13.x';
	T_MonitorByte2Name	:= '';
	T_Monitor2Bytes		:= FALSE;

	14:
	T_MonitorWord  		:= IW_64A1;
	T_MonitorByte1Name	:= 'IX14.x';
	T_MonitorByte2Name	:= '';
	T_Monitor2Bytes		:= FALSE;

	15:
	T_MonitorWord  		:= IW_65A1;
	T_MonitorByte1Name	:= 'IX15.x';
	T_MonitorByte2Name	:= '';
	T_Monitor2Bytes		:= FALSE;
	
	16:
	T_MonitorWord  		:= IW_66A1;
	T_MonitorByte1Name	:= 'IX16.x';
	T_MonitorByte2Name	:= '';
	T_Monitor2Bytes		:= FALSE;
	
	100:
	T_MonitorWord  		:= IW_141DI1;
	T_MonitorByte1Name	:= 'IX100.x';
	T_MonitorByte2Name	:= 'IX101.x';
	T_Monitor2Bytes		:= TRUE;

	110:
	T_MonitorWord  		:= IW_160A1;
	T_MonitorByte1Name	:= 'IX110.x';
	T_MonitorByte2Name	:= '';
	T_Monitor2Bytes		:= FALSE;

	111:
	T_MonitorWord  		:= IW_161A1;
	T_MonitorByte1Name	:= 'IX111.x';
	T_MonitorByte2Name	:= '';
	T_Monitor2Bytes		:= FALSE;

	112:
	T_MonitorWord  		:= IW_162A1;
	T_MonitorByte1Name	:= 'IX112.x';
	T_MonitorByte2Name	:= '';
	T_Monitor2Bytes		:= FALSE;
	
	113:
	T_MonitorWord  		:= IW_163A1;
	T_MonitorByte1Name	:= 'IX113.x';
	T_MonitorByte2Name	:= '';
	T_Monitor2Bytes		:= FALSE;

	200:
	T_MonitorWord  		:= IW_241DI1;
	T_MonitorByte1Name	:= 'IX200.x';
	T_MonitorByte2Name	:= 'IX201.x';
	T_Monitor2Bytes		:= TRUE;

	210:
	T_MonitorWord  		:= IW_260A1;
	T_MonitorByte1Name	:= 'IX210.x';
	T_MonitorByte2Name	:= 'IX211.x';
	T_Monitor2Bytes		:= FALSE;

(*		
	310:
	T_MonitorWord  		:= IW_260A1;
	T_MonitorByte1Name	:= 'IX200.x';
	T_MonitorByte2Name	:= 'IX201.x';
	T_Monitor2Bytes		:= TRUE;

	300:
	T_MonitorWord  		:= IW_341DI1;
	T_MonitorByte1Name	:= 'IX300.x';
	T_MonitorByte2Name	:= 'IX301.x';
	T_Monitor2Bytes		:= TRUE;

	310:
	T_MonitorWord  		:= IW_360A1;
	T_MonitorByte1Name	:= 'IX310.x';
	T_MonitorByte2Name	:= '';
	T_Monitor2Bytes		:= FALSE;

	311:
	T_MonitorWord  		:= IW_361A1	;
	T_MonitorByte1Name	:= 'IX311.x';
	T_MonitorByte2Name	:= '';
	T_Monitor2Bytes		:= FALSE;

	312:
	T_MonitorWord  		:= IW_362A1	;
	T_MonitorByte1Name	:= 'IX312.x';
	T_MonitorByte2Name	:= '';
	T_Monitor2Bytes		:= FALSE;

	313:
	T_MonitorWord  		:= QW_363A1	;
	T_MonitorByte1Name	:= 'QX310.x';
	T_MonitorByte2Name	:= '';
	T_Monitor2Bytes		:= FALSE;
	
	314:
	T_MonitorWord  		:= IW_364A1	;
	T_MonitorByte1Name	:= 'IX313.x';
	T_MonitorByte2Name	:= '';
	T_Monitor2Bytes		:= FALSE;
	
	315:
	T_MonitorWord  		:= QW_365A1	;
	T_MonitorByte1Name	:= 'QX311.x';
	T_MonitorByte2Name	:= '';
	T_Monitor2Bytes		:= FALSE;
*)
	
	1000:
	T_MonitorWord  		:= QW_41DO1;
	T_MonitorByte1Name	:= 'QX0.x';
	T_MonitorByte2Name	:= 'QX1.x';
	T_Monitor2Bytes		:= TRUE;

	1001:	
	T_MonitorWord  		:= QW_41DO2;
	T_MonitorByte1Name	:= 'QX2.x';
	T_MonitorByte2Name	:= 'QX3.x';
	T_Monitor2Bytes		:= TRUE;

	1050:
	T_MonitorWord  		:= QW_70A1;
	T_MonitorByte1Name	:= 'QX50.x';
	T_MonitorByte2Name	:= 'QX51.x';
	T_Monitor2Bytes		:= TRUE;
	
	1051:
	T_MonitorWord  		:= QW_70A1_0;
	T_MonitorByte1Name	:= 'QX52.x';
	T_MonitorByte2Name	:= 'QX53.x';
	T_Monitor2Bytes		:= FALSE;

	1060:
	T_MonitorWord  		:= QW_71A1;
	T_MonitorByte1Name	:= 'QX60.x';
	T_MonitorByte2Name	:= 'QX61.x';
	T_Monitor2Bytes		:= TRUE;
	
	1100:
	T_MonitorWord  		:= QW_141DO1;
	T_MonitorByte1Name	:= 'QX100.x';
	T_MonitorByte2Name	:= 'QX101.x';
	T_Monitor2Bytes		:= TRUE;

	1150:
	T_MonitorWord  		:= QW_170A1;
	T_MonitorByte1Name	:= 'QX150.x';
	T_MonitorByte2Name	:= 'QX151.x';
	T_Monitor2Bytes		:= TRUE;

	1200:
	T_MonitorWord  		:= QW_241DO1	;
	T_MonitorByte1Name	:= 'QX200.x';
	T_MonitorByte2Name	:= 'QX201.x';
	T_Monitor2Bytes		:= TRUE;
(*	
	1300:
	T_MonitorWord  		:= QW_341DO1;
	T_MonitorByte1Name	:= 'QX300.x';
	T_MonitorByte2Name	:= 'QX301.x';
	T_Monitor2Bytes		:= TRUE;
*)
	1350:
	T_MonitorWord  		:= QW_350A1;
	T_MonitorByte1Name	:= 'QX350.x';
	T_MonitorByte2Name	:= 'QX351.x';
	T_Monitor2Bytes		:= TRUE;
	
	
END_CASE


(********************** Machine Speed Override *****************************)
IF HMI.V_MachineSpeed <= 10 THEN 
	HMI.V_MachineSpeed :=10;	
END_IF

END_PROGRAM

// ---- POUs/MC/Statistic.TcPOU
PROGRAM Statistic
VAR
	pls_1Minute			:BOOL;	
	tmr_1Minute			:TON;
	pls_1Second			:BOOL;	
	tmr_1Second			:TON;
	plsReportDone			:F_TRIG;
	plsServiceStop			:R_Trig;
	plsGlueL_Shift			:R_Trig;
	plsTapeL_Shift			:R_trig;
	plsGlueL_All			:R_Trig;
	plsTapeL_All			:R_trig;	
	plsGlueR_Shift			:R_Trig;
	plsTapeR_Shift			:R_trig;
	plsGlueR_All			:R_Trig;
	plsTapeR_All			:R_trig;		
	
	LocalSystemTime		:FB_LocalSystemTime;
	Current_Date		:STRING;	
	
	RunStep_Report		:INT;
	WeekDay				:STRING;
	ProdSpd_Efficiency	:REAL;
	ProdSpd_OEE			:REAL;
	
END_VAR

// *************************************************
(* Timer Pulse *)
tmr_1Minute(IN:= NOT pls_1Minute , PT:= T#60S);
pls_1Minute := tmr_1Minute.Q;
tmr_1Second(IN:= NOT pls_1Second , PT:= T#1S);
pls_1Second := tmr_1Second.Q;


(* PC Local Time *)
LocalSystemTime(
	sNetID:= '10.1.33.138.1.1' , 
	bEnable:= TRUE , 
	dwCycle:= , 
	dwOpt:= , 
	tTimeout:= , 
	bValid=> , 
	systemTime=> , 
	tzID=> );

(* Weekday *)
CASE LocalSystemTime.systemTime.wDayOfWeek OF
	0: WeekDay := 'SUN'	;
	1: WeekDay := 'MON'	;
	2: WeekDay := 'TUE'	;
	3: WeekDay := 'WED'	;
	4: WeekDay := 'THUR';
	5: WeekDay := 'FRI'	;
	6: WeekDay := 'SAT'	;					
END_CASE
	
// *************************************************************
(*	To Calculate Current Shift Number	*)
IF LocalSystemTime.systemTime.wYear <> 1970 THEN
IF 	(WORD_TO_UINT(LocalSystemTime.systemTime.wHour) 	> Statistic_Shift_StartTimeH[1] OR
	(WORD_TO_UINT(LocalSystemTime.systemTime.wHour) 	= Statistic_Shift_StartTimeH[1] AND LocalSystemTime.systemTime.wMinute 	>= Statistic_Shift_StartTimeM[1]) )
	AND
	(WORD_TO_UINT(LocalSystemTime.systemTime.wHour) 	< Statistic_Shift_EndTimeH[1] OR
	(WORD_TO_UINT(LocalSystemTime.systemTime.wHour) 	= Statistic_Shift_EndTimeM[1] AND LocalSystemTime.systemTime.wMinute 	<= Statistic_Shift_EndTimeM[1]))
THEN
	Statistic_CurShift_Number := 1;
ELSE	
		IF 	(WORD_TO_UINT(LocalSystemTime.systemTime.wHour) 	> Statistic_Shift_StartTimeH[2] OR
			(WORD_TO_UINT(LocalSystemTime.systemTime.wHour) 	= Statistic_Shift_StartTimeH[2] AND LocalSystemTime.systemTime.wMinute 	>= Statistic_Shift_StartTimeM[2]) )
			AND
			(WORD_TO_UINT(LocalSystemTime.systemTime.wHour) 	< Statistic_Shift_EndTimeH[2] OR
			(WORD_TO_UINT(LocalSystemTime.systemTime.wHour) 	= Statistic_Shift_EndTimeM[2] AND LocalSystemTime.systemTime.wMinute 	<= Statistic_Shift_EndTimeM[2]))
		THEN
			Statistic_CurShift_Number := 2;
ELSE	
		IF 	(WORD_TO_UINT(LocalSystemTime.systemTime.wHour) 	> Statistic_Shift_StartTimeH[3] OR
			(WORD_TO_UINT(LocalSystemTime.systemTime.wHour) 	= Statistic_Shift_StartTimeH[3] AND LocalSystemTime.systemTime.wMinute 	>= Statistic_Shift_StartTimeM[3]) )
			AND
			(WORD_TO_UINT(LocalSystemTime.systemTime.wHour) 	< Statistic_Shift_EndTimeH[3] OR
			(WORD_TO_UINT(LocalSystemTime.systemTime.wHour) 	= Statistic_Shift_EndTimeM[3] AND LocalSystemTime.systemTime.wMinute 	<= Statistic_Shift_EndTimeM[3]))
		THEN
					Statistic_CurShift_Number := 3;
		ELSE				
					Statistic_CurShift_Number := 0;
END_IF
END_IF					
END_IF
END_IF

// ***********************************************************************************************
(* Generate Report *)
CASE RunStep_Report OF
	0: (* To check shift number change *)
		IF 	(Statistic_PreviousShift_Number <> Statistic_CurShift_Number) THEN
			RunStep_Report	:= RunStep_Report + 10;		
		END_IF
	
	10: (* Copy Statistic to History for Reporting then reset current shift data *)
		Statistic_History	:= Statistic_Current;
(* Date *)		
		Statistic_Current.ShiftInformation	:= WORD_TO_STRING(LocalSystemTime.systemTime.wDay) ;
		Statistic_Current.ShiftInformation	:=	CONCAT(STR1:= Statistic_Current.ShiftInformation , STR2:= '-' );
		Statistic_Current.ShiftInformation	:=	CONCAT(STR1:= Statistic_Current.ShiftInformation , STR2:= WORD_TO_STRING(LocalSystemTime.systemTime.wMonth ));
		Statistic_Current.ShiftInformation	:=	CONCAT(STR1:= Statistic_Current.ShiftInformation , STR2:= '-' );
		Statistic_Current.ShiftInformation	:=	CONCAT(STR1:= Statistic_Current.ShiftInformation , STR2:= WORD_TO_STRING(LocalSystemTime.systemTime.wYear ));
		Statistic_Current.ShiftInformation	:=	CONCAT(STR1:= Statistic_Current.ShiftInformation , STR2:= ' ' );
		Statistic_Current.ShiftInformation	:=	CONCAT(STR1:= Statistic_Current.ShiftInformation , STR2:= WeekDay );		
		Statistic_Current.ShiftInformation	:=	CONCAT(STR1:= Statistic_Current.ShiftInformation , STR2:= ' - ' );
(* Start Time *)		
		IF Statistic_Shift_StartTimeH[Statistic_CurShift_Number] < 10 THEN
			Statistic_Current.ShiftInformation	:=	CONCAT(STR1:= Statistic_Current.ShiftInformation , STR2:= '0' );
		END_IF
		Statistic_Current.ShiftInformation	:=	CONCAT(STR1:= Statistic_Current.ShiftInformation , STR2:= WORD_TO_STRING(Statistic_Shift_StartTimeH[Statistic_CurShift_Number] ));
		IF Statistic_Shift_StartTimeM[Statistic_CurShift_Number] < 10 THEN
			Statistic_Current.ShiftInformation	:=	CONCAT(STR1:= Statistic_Current.ShiftInformation , STR2:= '0' );
		END_IF
		Statistic_Current.ShiftInformation	:=	CONCAT(STR1:= Statistic_Current.ShiftInformation , STR2:= WORD_TO_STRING(Statistic_Shift_StartTimeM[Statistic_CurShift_Number] ));
		
		Statistic_Current.ShiftInformation	:=	CONCAT(STR1:= Statistic_Current.ShiftInformation , STR2:= ' - ' );
(* End Time *)
		IF Statistic_Shift_EndTimeH[Statistic_CurShift_Number] < 10 THEN
			Statistic_Current.ShiftInformation	:=	CONCAT(STR1:= Statistic_Current.ShiftInformation , STR2:= '0' );
		END_IF
		Statistic_Current.ShiftInformation	:=	CONCAT(STR1:= Statistic_Current.ShiftInformation , STR2:= WORD_TO_STRING(Statistic_Shift_EndTimeH[Statistic_CurShift_Number] ));
		IF Statistic_Shift_EndTimeM[Statistic_CurShift_Number] < 10 THEN
			Statistic_Current.ShiftInformation	:=	CONCAT(STR1:= Statistic_Current.ShiftInformation , STR2:= '0' );
		END_IF
		Statistic_Current.ShiftInformation	:=	CONCAT(STR1:= Statistic_Current.ShiftInformation , STR2:= WORD_TO_STRING(Statistic_Shift_EndTimeM[Statistic_CurShift_Number] ));

(* Reset Data *)
		Statistic_Current.RejectLeftTape		:= 0;
		Statistic_Current.RejectRightTape		:= 0;
		Statistic_Current.RejectUnderWeight		:= 0;
		Statistic_Current.RejectOverWeight		:= 0;
		Statistic_Current.GoodCase				:= 0;
		Statistic_Current.RunTime_Second		:= 0;
		Statistic_Current.ExternalStop_Second	:= 0;
		Statistic_Current.InternalStop_Second	:= 0;
		Statistic_Current.WaitingTime_Second	:= 0;
		Statistic_Current.RejectCaseRemoved		:= 0;
		Statistic_Current.ServiceStop_Number	:= 0;	
		Statistic_Current.ServiceStop_Second	:= 0;
		Statistic_Current.StackerFault_Number	:= 0;
		Statistic_Current.StackerFault_Second	:= 0;
		Statistic_Current.XPusherFault_Number	:= 0;
		Statistic_Current.XPusherFault_Second	:= 0;
		Statistic_Current.YPusherFault_Number	:= 0;
		Statistic_Current.YPusherFault_Second	:= 0;
		Statistic_Current.ErectorFault_Number	:= 0;
		Statistic_Current.ErectorFault_Second	:= 0;
		Statistic_Current.ExitFault_Number		:= 0;
		Statistic_Current.ExitFault_Second		:= 0;
		Statistic_Current.HorizontalFault_Number:= 0;
		Statistic_Current.HorizontalFault_Second:= 0;
		Statistic_Current.MajorFault_Number		:= 0;
		Statistic_Current.MajorFault_Second		:= 0;			
		Statistic_Current.GlueLeft_Number		:= 0;	
		Statistic_Current.GlueRight_Number		:= 0;			
		Statistic_Current.TapeLeft_Number		:= 0;	
		Statistic_Current.TapeRight_Number		:= 0;				
		Statistic_Current.RecipeName			:= CurrRecipe.sDescription;
		
		RunStep_Report	:= RunStep_Report + 10;	
		
	20: (* To Generate Report *)
		IF	(Statistic_PreviousShift_Number <>0) THEN
			Generate_Report	:=1;
		END_IF	
			Statistic_PreviousShift_Number	:=Statistic_CurShift_Number;
			RunStep_Report	:= RunStep_Report + 10;	
			
	30: (* Waiting for Reporting Done *)		
		IF NOT Generate_Report THEN
			RunStep_Report	:= 0;
		END_IF
END_CASE

// **********************************************************************************************************
(* Production Data Update *)
IF (Statistic_Current.GoodCase + 
	Statistic_Current.RejectLeftTape + 
	Statistic_Current.RejectRightTape + 
	Statistic_Current.RejectOverWeight + 
	Statistic_Current.RejectUnderWeight + 
	Statistic_Current.RejectCaseRemoved ) > 0 THEN
	Statistic_Current.Production_Percentage	:= 	DINT_TO_REAL(Statistic_Current.GoodCase * 100) / 
												DINT_TO_REAL((Statistic_Current.GoodCase + 
												Statistic_Current.RejectLeftTape + 
												Statistic_Current.RejectRightTape +
												Statistic_Current.RejectOverWeight +
												Statistic_Current.RejectUnderWeight +
												Statistic_Current.RejectCaseRemoved));
											
	Statistic_Current.Reject_Percentage		:= 	DINT_TO_REAL((Statistic_Current.RejectLeftTape + 
												Statistic_Current.RejectRightTape +
												Statistic_Current.RejectOverWeight +
												Statistic_Current.RejectUnderWeight +
												Statistic_Current.RejectCaseRemoved ) * 100)/
												DINT_TO_REAL((Statistic_Current.GoodCase + 
												Statistic_Current.RejectLeftTape + 
												Statistic_Current.RejectRightTape +
												Statistic_Current.RejectOverWeight +
												Statistic_Current.RejectUnderWeight +
												Statistic_Current.RejectCaseRemoved));
				
ELSE
	Statistic_Current.Production_Percentage	:= 0;
	Statistic_Current.Reject_Percentage		:= 0;
END_IF											


							
IF (Statistic_Current.RunTime_Second + Statistic_Current.ExternalStop_Second + Statistic_Current.InternalStop_Second + Statistic_Current.WaitingTime_Second)>0 THEN
	ProdSpd_Efficiency					:= 	DINT_TO_REAL(Cfg_prodSpeed_perHour)/3600 *	
											DINT_TO_REAL(Statistic_Current.RunTime_Second + Statistic_Current.ExternalStop_Second + Statistic_Current.InternalStop_Second + Statistic_Current.WaitingTime_Second);
	Statistic_Current.Net_Efficiency	:= Statistic_Current.GoodCase * 100 / ProdSpd_Efficiency;											
ELSE
	ProdSpd_Efficiency					:= 0;
	Statistic_Current.Net_Efficiency	:= 0;
END_IF	

IF (Statistic_Current.RunTime_Second + Statistic_Current.InternalStop_Second)>0 THEN											
	ProdSpd_OEE							:= 	DINT_TO_REAL(Cfg_prodSpeed_perHour)/3600 *		
										 	DINT_TO_REAL(Statistic_Current.RunTime_Second + Statistic_Current.InternalStop_Second);
	Statistic_Current.OEE				:= Statistic_Current.GoodCase * 100 / ProdSpd_OEE;
ELSE
	ProdSpd_OEE							:=0;
	Statistic_Current.OEE				:=0;
END_IF

// *************************************************************************************************
// To set fault statistic memory
IF 		NOT H_ServiceStop_Pressed 
	AND NOT MajorFault_Triggered 
	AND NOT StackerFault_Triggered 
	AND NOT XPusherFault_Triggered 
	AND NOT YPusherFault_Triggered 
	AND NOT ErectorFault_Triggered
	AND NOT ExitFault_Triggered
	AND NOT HorizontalFault_Triggered	THEN
	
	IF 		mc.Trouble	THEN
			MajorFault_Triggered					:= TRUE;
			Statistic_Current.MajorFault_Number		:= Statistic_Current.MajorFault_Number + 1;
			Statistic_Manual.MajorFault_Number		:= Statistic_Manual.MajorFault_Number + 1;
			Statistic_Total.MajorFault_Number		:= Statistic_Total.MajorFault_Number + 1;
	ELSIF	SC[0].MinorFault THEN
			StackerFault_Triggered 					:= TRUE;	
			Statistic_Current.StackerFault_Number	:= Statistic_Current.StackerFault_Number + 1;
			Statistic_Manual.StackerFault_Number	:= Statistic_Manual.StackerFault_Number + 1;
			Statistic_Total.StackerFault_Number		:= Statistic_Total.StackerFault_Number + 1;
	ELSIF 	SC[1].MinorFault THEN
			XPusherFault_Triggered					:= TRUE;
			Statistic_Current.XPusherFault_Number	:= Statistic_Current.XPusherFault_Number + 1;
			Statistic_Manual.XPusherFault_Number	:= Statistic_Manual.XPusherFault_Number + 1;
			Statistic_Total.XPusherFault_Number		:= Statistic_Total.XPusherFault_Number + 1;
	ELSIF 	SC[2].MinorFault THEN
			YPusherFault_Triggered					:= TRUE;
			Statistic_Current.YPusherFault_Number	:= Statistic_Current.YPusherFault_Number + 1;
			Statistic_Manual.YPusherFault_Number	:= Statistic_Manual.YPusherFault_Number + 1;
			Statistic_Total.YPusherFault_Number		:= Statistic_Total.YPusherFault_Number + 1;			
	ELSIF 	SC[3].MinorFault THEN
			ErectorFault_Triggered					:= TRUE;
			Statistic_Current.ErectorFault_Number	:= Statistic_Current.ErectorFault_Number + 1;
			Statistic_Manual.ErectorFault_Number	:= Statistic_Manual.ErectorFault_Number + 1;
			Statistic_Total.ErectorFault_Number		:= Statistic_Total.ErectorFault_Number + 1;				
	ELSIF 	SC[4].MinorFault THEN
			ExitFault_Triggered						:= TRUE;
			Statistic_Current.ExitFault_Number		:= Statistic_Current.ExitFault_Number + 1;
			Statistic_Manual.ExitFault_Number		:= Statistic_Manual.ExitFault_Number + 1;
			Statistic_Total.ExitFault_Number		:= Statistic_Total.ExitFault_Number + 1;		
	ELSIF 	SC[6].MinorFault THEN
			HorizontalFault_Triggered				:= TRUE;
			Statistic_Current.HorizontalFault_Number:= Statistic_Current.HorizontalFault_Number + 1;
			Statistic_Manual.HorizontalFault_Number	:= Statistic_Manual.HorizontalFault_Number + 1;
			Statistic_Total.HorizontalFault_Number	:= Statistic_Total.HorizontalFault_Number + 1;				
	END_IF
END_IF

// ************************************************************************************************											
(* Update Statistic Data by Timer *)
IF pls_1Second THEN
// During shift
	IF Statistic_CurShift_Number >0 THEN
		IF 	H_ServiceStop_Pressed THEN
			Statistic_Current.ServiceStop_Second := Statistic_Current.ServiceStop_Second + 1;
		END_IF	
		IF MajorFault_Triggered THEN
			Statistic_Current.MajorFault_Second		:= Statistic_Current.MajorFault_Second + 1;			
		END_IF
		IF StackerFault_Triggered THEN
			Statistic_Current.StackerFault_Second	:= Statistic_Current.StackerFault_Second + 1;			
		END_IF
		IF XPusherFault_Triggered THEN
			Statistic_Current.XPusherFault_Second	:= Statistic_Current.XPusherFault_Second + 1;			
		END_IF
		IF YPusherFault_Triggered THEN
			Statistic_Current.YPusherFault_Second	:= Statistic_Current.YPusherFault_Second + 1;			
		END_IF
		IF ErectorFault_Triggered THEN
			Statistic_Current.ErectorFault_Second	:= Statistic_Current.ErectorFault_Second + 1;			
		END_IF
		IF ExitFault_Triggered THEN
			Statistic_Current.ExitFault_Second		:= Statistic_Current.ExitFault_Second + 1;			
		END_IF
		IF HorizontalFault_Triggered THEN
			Statistic_Current.HorizontalFault_Second:= Statistic_Current.HorizontalFault_Second + 1;			
		END_IF
	
		
		IF mc.Trouble OR mc.StationStopErr OR NOT mc.AutoRunning THEN
			Statistic_Current.InternalStop_Second	:= Statistic_Current.InternalStop_Second + 1;
		ELSIF 	CO_YPush_Auto.YWaitingTime.Q THEN
			Statistic_Current.WaitingTime_Second	:= Statistic_Current.WaitingTime_Second + 1;
		ELSE
			Statistic_Current.RunTime_Second		:= Statistic_Current.RunTime_Second + 1;
		END_IF

	END_IF

// All Time	
		IF 	H_ServiceStop_Pressed THEN
			Statistic_Total.ServiceStop_Second := Statistic_Total.ServiceStop_Second + 1;
			Statistic_Manual.ServiceStop_Second := Statistic_Manual.ServiceStop_Second + 1;
		END_IF	
		IF MajorFault_Triggered THEN
			Statistic_Total.MajorFault_Second		:= Statistic_Total.MajorFault_Second + 1;	
			Statistic_Manual.MajorFault_Second		:= Statistic_Manual.MajorFault_Second + 1;			
		END_IF
		IF StackerFault_Triggered THEN
			Statistic_Total.StackerFault_Second		:= Statistic_Total.StackerFault_Second + 1;	
			Statistic_Manual.StackerFault_Second	:= Statistic_Manual.StackerFault_Second + 1;			
		END_IF
		IF XPusherFault_Triggered THEN
			Statistic_Total.XPusherFault_Second		:= Statistic_Total.XPusherFault_Second + 1;	
			Statistic_Manual.XPusherFault_Second	:= Statistic_Manual.XPusherFault_Second + 1;					
		END_IF
		IF YPusherFault_Triggered THEN
			Statistic_Total.YPusherFault_Second		:= Statistic_Total.YPusherFault_Second + 1;	
			Statistic_Manual.YPusherFault_Second	:= Statistic_Manual.YPusherFault_Second + 1;			
		END_IF
		IF ErectorFault_Triggered THEN
			Statistic_Total.ErectorFault_Second		:= Statistic_Total.ErectorFault_Second + 1;		
			Statistic_Manual.ErectorFault_Second	:= Statistic_Manual.ErectorFault_Second + 1;		
		END_IF
		IF ExitFault_Triggered THEN
			Statistic_Total.ExitFault_Second		:= Statistic_Total.ExitFault_Second + 1;		
			Statistic_Manual.ExitFault_Second		:= Statistic_Manual.ExitFault_Second + 1;		
		END_IF
		IF HorizontalFault_Triggered THEN
			Statistic_Total.HorizontalFault_Second	:= Statistic_Total.HorizontalFault_Second + 1;	
			Statistic_Manual.HorizontalFault_Second	:= Statistic_Manual.HorizontalFault_Second + 1;			
		END_IF
		
		IF mc.Trouble OR mc.StationStopErr OR NOT mc.AutoRunning THEN
			Statistic_Total.InternalStop_Second		:= Statistic_Total.InternalStop_Second + 1;
			Statistic_Manual.InternalStop_Second	:= Statistic_Manual.InternalStop_Second + 1;			
		ELSIF 	CO_YPush_Auto.YWaitingTime.Q THEN
			Statistic_Total.WaitingTime_Second		:= Statistic_Total.WaitingTime_Second + 1;
			Statistic_Manual.WaitingTime_Second		:= Statistic_Manual.WaitingTime_Second + 1;			
		ELSE
			Statistic_Total.RunTime_Second			:= Statistic_Total.RunTime_Second + 1;
			Statistic_Manual.RunTime_Second			:= Statistic_Manual.RunTime_Second + 1;			
	END_IF	
	
END_IF

// **************************************************************************************************
(* Update Statistic Data by Counter *)
plsServiceStop	(CLK:= H_ServiceStop_Pressed);
IF plsServiceStop.Q THEN
Statistic_Current.ServiceStop_Number	:= Statistic_Current.ServiceStop_Number + 1;
END_IF

IF Statistic_CurShift_Number >0 THEN
		plsGlueL_Shift	(CLK:= O_Nord_ValveL_On);
		IF plsGlueL_Shift.Q THEN
			Statistic_Current.GlueLeft_Number := Statistic_Current.GlueLeft_Number + 1;
		END_IF
		plsTapeL_Shift	(CLK:=I_HOR_TapeL_Empty_PE);	
		IF plsTapeL_Shift.Q THEN
			Statistic_Current.TapeLeft_Number := Statistic_Current.TapeLeft_Number + 1;
		END_IF	
		plsGlueR_Shift	(CLK:= O_Nord_ValveR_On);
		IF plsGlueR_Shift.Q THEN
			Statistic_Current.GlueRight_Number := Statistic_Current.GlueRight_Number + 1;
		END_IF		
		plsTapeR_Shift	(CLK:=I_HOR_TapeR_Empty_PE);	
		IF plsTapeR_Shift.Q THEN
			Statistic_Current.TapeRight_Number := Statistic_Current.TapeRight_Number + 1;
		END_IF	
END_IF

END_PROGRAM

// ---- POUs/Collator/Y Pusher n Bridge/CO_YPush_Auto.TcPOU
PROGRAM CO_YPush_Auto
VAR_IN_OUT
	Station		:structStationCtrl;
END_VAR
VAR
	Timeout:ton;
	ManualInit_TOn:Ton;
	CO_YStk_AtBuf1_PEOff_Ton : ton;
	TimeoutTrigger	: BOOL;
	PTC_OK			: BOOL;
	TimeoutSetting	: TIME;
	
	BundleFull		:BOOL;
	NoBundle		:BOOL;
	YWaitingTime	:Ton;
END_VAR

CurrRecipe.iStackX	:= 6;

CASE CurrRecipe.iStackX OF
	1:
		PTC_OK := I_CO_PTC_PE1;
	2:
		PTC_OK := I_CO_PTC_PE1 AND I_CO_PTC_PE2;
	3:
		PTC_OK := I_CO_PTC_PE1 AND I_CO_PTC_PE2 AND I_CO_PTC_PE3;
	4:
		PTC_OK := I_CO_PTC_PE1 AND I_CO_PTC_PE2 AND I_CO_PTC_PE3 AND I_CO_PTC_PE4;
	5:
		PTC_OK := I_CO_PTC_PE1 AND I_CO_PTC_PE2 AND I_CO_PTC_PE3 AND I_CO_PTC_PE4 AND I_CO_PTC_PE5;
	6:
		PTC_OK := I_CO_PTC_PE1 AND I_CO_PTC_PE2 AND I_CO_PTC_PE3 AND I_CO_PTC_PE4 AND I_CO_PTC_PE5 AND I_CO_PTC_PE6;
	7:
		PTC_OK := I_CO_PTC_PE1 AND I_CO_PTC_PE2 AND I_CO_PTC_PE3 AND I_CO_PTC_PE4 AND I_CO_PTC_PE5 AND I_CO_PTC_PE6 AND I_CO_PTC_PE7;
	8:
		PTC_OK := I_CO_PTC_PE1 AND I_CO_PTC_PE2 AND I_CO_PTC_PE3 AND I_CO_PTC_PE4 AND I_CO_PTC_PE5 AND I_CO_PTC_PE6 AND I_CO_PTC_PE7 AND I_CO_PTC_PE8;
		
	ELSE
		PTC_OK := FALSE;												
END_CASE

YWaitingTime	(In:= NOT PTC_OK, PT:= T#5S);

(**************************************************************************************************************)
(* GENERAL STATION MAPPING  *)
(**************************************************************************************************************)
Station.Name			:=	'COLLATOR Y PUSHER AND BRIDGE';
Station.Rdy 			:= 	Station.Origin;
Station.AutoRun 		:=	(MC.AutoRunning OR Station.M_Step) AND 
							NOT (Station.Bypass OR Station.MajorFault OR Station.MinorFault);
Station.RunReq			:= 	((H_CO_StkRdyForYPush  OR mc.DryRun) 
							AND(NOT (H_ER_CtnSideFlapDone OR H_ER_CtnPushInDone)))
							OR Station.M_Step ;
Station.RunCond			:=	(NOT ER.Running OR ER.RunStep >= 20) AND(*Erector Arm Not Running*)
							NOT (Station.Done OR MC.StopPressed);
Station.Run_NextStepPls	:=	(Station.AutoRun AND NOT Station.M_Step) OR 
							(Station.M_Step AND M_StepFwdPls) OR HMI.T_OneCycleRun;
Station.Run_PrevStepPls	:=	(Station.M_Step AND M_StepBwdPls);

(**************************************************************************************************************)
(*	Initial Device	, detect there is a cartoon *)
(**************************************************************************************************************)

IF CO_Bdl_Reach_TON.Q THEN
	H_CO_StkRdyForYPush := TRUE;
END_IF


(**************************************************************************************************************)
(*	Initial Device	*)
(**************************************************************************************************************)
ManualInit_TOn (in:= mc.ManualMode AND NOT mc.OriginSchRun, pt:= T#1S);

IF mc.ManualMode AND NOT mc.OriginSchRun AND NOT ManualInit_TOn.Q THEN
	CO_YPush_Srv_Var.In_MoveAbs := FALSE;
END_IF

(**************************************************************************************************************)
(* Auto Sequance*)
(**************************************************************************************************************)

TimeoutSetting	:= T#50S;
Timeout(IN:=TimeoutTrigger, PT:=TimeoutSetting);
IF Timeout.Q THEN
	TimeoutTrigger := FALSE;
END_IF
CO_YStk_AtBuf1_PEOff_Ton ( IN:= (Station.RunStep = 0) AND NOT I_CO_YStk_AtBuf1_PE , pt:= T#3S);

IF Station.AutoRun OR Station.M_Step THEN
	
	CASE Station.RunStep OF

	0 : 	(************* Ready To Run ****************)
			IF Station.RunCond AND Station.RunReq AND Station.Rdy THEN
				IF BundleFull OR mc.DryRun OR NOT Cfg_EnbAutoWA	THEN
					IF (H_ER_CtnRdyForPushIn AND NOT H_ER_CtnPushInDone) OR 
						Station.M_Step OR Cfg_BypassErector THEN
						Station.RunStep := 100;
					END_IF
				ELSE	
					E_PTC_BundleNOK			:= TRUE;
					Station.SeqFaultString 	:= 'Auto: Part Transfer Confirmation Not Complete';				
				END_IF
				
			ELSIF H_CO_StkRdyForYPush AND CO_YStk_AtBuf1_PEOff_Ton.Q AND NOT mc.DryRun  THEN
				Station.SeqFaultWord 	:= 200;
				E_Buf1_BundleMissing	:= TRUE;	
				Station.SeqFaultString 	:= 'Auto: Stack Missing at Buffer 1 Area.';										
			ELSIF NOT Station.RunCond THEN
				Station.Status 			:= '0: Station Waiting for Run Conditions';
				Station.StatusInt		:= 1;
			ELSIF NOT Station.RunReq THEN
				Station.Status 			:= '0: Station Waiting for Run Request';
				Station.StatusInt		:= 2;
			ELSE
				Station.Status 			:= '0: Station Not Ready';	
				Station.StatusInt		:= 3;			
			END_IF
	
	100 : 	(************* Bridge Cylinder, Flap Guides Forward ****************)
			Station.Status 		:= '100: Bridge Cylinders & Flap Guides Forward';
			Station.StatusInt	:= 152;
			
			CO_Brdg_Cyl_Var.In_AutoWork := TRUE;
			CO_Brdg_Cyl_Var.In_AutoHome := FALSE;

			CO_FlapGuide_Cyl_Var.In_AutoWork := TRUE;
			CO_FlapGuide_Cyl_Var.In_AutoHome := FALSE;
			
			CO_YPush_Cyl_Var.In_AutoWork := FALSE;
			CO_YPush_Cyl_Var.In_AutoHome := TRUE;

			
			CO_YPush_Srv_Var.In_PosCmd := H_CO_YPush_Srv_CtnFinalPos;
			CO_YPush_Srv_Var.In_VelCmd := A_Srv_YPusherLoSpeed;
			IF 	CO_YPush_Srv_Var.In_MoveXLock 		AND 
				CO_Brdg_Cyl_Var.In_WorkXLock 		AND 
				NOT CO_Brdg_Cyl_Var.S_HomePos		AND 
				NOT CO_FlapGuide_Cyl_Var.S_HomePos 	
				AND CO_YPush_Cyl_Var.S_HomePos		THEN
				CO_YPush_Srv_Var.In_MoveAbs := TRUE;
				CO_YPush_Cyl_Var.In_AutoWork := FALSE;
				CO_YPush_Cyl_Var.In_AutoHome := FALSE;			
			END_IF
		
			IF 	CO_Brdg_Cyl_Var.S_WorkPos 		AND 
				CO_FlapGuide_Cyl_Var.S_WorkPos 	AND
				Station.Run_NextStepPls 		THEN
				CO_YPush_Srv_Var.In_MoveAbs := FALSE;
				CO_Brdg_Cyl_Var.In_AutoWork := FALSE;
				CO_FFlapBrdg_Cyl_Var.In_AutoWork := FALSE;
				CO_FlapGuide_Cyl_Var.In_AutoWork := FALSE;
				Station.RunStep := Station.RunStep + 10;
			END_IF
			

	110 : 	(************* Move Y Pusher To Push Stack into Carton  ****************)
			Station.Status 		:= '110: Move Y Pusher To Push Stack into Carton';
			Station.StatusInt	:= 153;
			
			CO_YPush_Srv_Var.In_PosCmd := H_CO_YPush_Srv_CtnFinalPos;
			CO_YPush_Srv_Var.In_VelCmd := A_Srv_YPusherLoSpeed;
			CO_YPush_Srv_Var.In_MoveAbs := TRUE;

			
			IF 	CO_YPush_Srv_Var.Out_CurrPos >= (CO_YPush_Srv_Var.In_PosCmd - 100) THEN
				CO_YPush_Strk_Cyl_Var.In_AutoWork := TRUE;
				CO_YPush_Strk_Cyl_Var.In_AutoHome := FALSE;
			END_IF
			
			IF ((fcComparePos(CurrPos:= CO_YPush_Srv_Var.Out_CurrPos, TargetPos:= CO_YPush_Srv_Var.In_PosCmd, Tolerance := 0.5)) AND
							CO_YPush_Srv_Var.Out_InPos) AND
				CO_YPush_Strk_Cyl_Var.S_WorkPos AND
				Station.Run_NextStepPls THEN	
				H_CO_StkRdyForYPush := FALSE;	
				H_CO_Bdl_StkY_Count := 0;	
				CO_YPush_Srv_Var.In_MoveAbs := FALSE;
				CO_YPush_Strk_Cyl_Var.In_AutoWork := FALSE;
				
				IF NOT Cfg_BypassErector AND H_ER_CtnRdyForPushIn THEN
					H_ER_CtnPushInDone := TRUE;
				END_IF
				H_ER_CtnRdyForPushIn := FALSE;
				
				IF 	I_CO_YStk_AtBuf1_PE  THEN	
					Station.SeqFaultWord 	:= 204;	
					E_Buf1_BundleJam		:= TRUE;
					Station.SeqFaultString 	:= 'Auto: Stack Detected at Buffer 1 After Push. ';	
				ELSIF 	I_CO_YStk_AtBuf2_PE   THEN
					Station.SeqFaultWord 	:= 205;	
					E_Buf2_Sensor			:= TRUE;
					Station.SeqFaultString 	:= 'Auto: Stack Detected at Buffer 2 After Push. ';	
				ELSE
					Station.RunStep := Station.RunStep + 10;
				END_IF	
			END_IF

	115:	(************* Y Pusher Servo Move to Safe Pos ****************)			

			CO_YPush_Strk_Cyl_Var.In_AutoWork 	:= FALSE;
			CO_YPush_Strk_Cyl_Var.In_AutoHome 	:= TRUE;

				CO_YPush_Srv_Var.In_PosCmd := H_CO_YPush_Srv_SafePosition; 
				CO_YPush_Srv_Var.In_VelCmd := A_Srv_BeltAutoHiSpeed;
				CO_YPush_Srv_Var.In_MoveAbs := TRUE;
			
			
			IF ((fcComparePos(CurrPos:= CO_YPush_Srv_Var.Out_CurrPos, TargetPos:= H_CO_YPush_Srv_SafePosition, Tolerance := 0.5)) AND
			CO_YPush_Srv_Var.Out_InPos) AND  CO_YPush_Strk_Cyl_Var.S_HomePos THEN
			CO_YPush_Cyl_Var.In_AutoWork 		:= TRUE;
			CO_YPush_Cyl_Var.In_AutoHome 		:= FALSE;
				CO_YPush_Srv_Var.In_MoveAbs := FALSE;
			Station.RunStep := Station.RunStep+5;	
			END_IF


			
	120 : 	(************* Move Y Pusher Back To Home Position and all Cylinders Bwd  ****************)
			(************* Flap Guide Cylinder Bwd ****************)
			Station.Status 		:= '120: Move Y Pusher Back and all Cylinders Bwd';
			Station.StatusInt	:= 154;
				
			CO_Brdg_Cyl_Var.In_AutoWork 		:= FALSE;
			CO_Brdg_Cyl_Var.In_AutoHome			:= TRUE;
			CO_YPush_Strk_Cyl_Var.In_AutoWork 	:= FALSE;
			CO_YPush_Strk_Cyl_Var.In_AutoHome 	:= TRUE;		
			
			(* Temporary to test Push in and Out without lifting up Y-Pusher *)	
			CO_YPush_Srv_Var.In_PosCmd := H_CO_YPush_Srv_CurrStandbyPos;
			CO_YPush_Srv_Var.In_VelCmd := A_Srv_YPusherHiSpeed;
			CO_YPush_Srv_Var.In_MoveAbs := TRUE;
				
	(*		
			IF CO_YPush_Strk_Cyl_Var.S_HomePos THEN
				CO_YPush_Cyl_Var.In_AutoWork 		:= TRUE;
				CO_YPush_Cyl_Var.In_AutoHome 		:= FALSE;
			END_IF
	*)		
			IF	 CO_YPush_Cyl_Var.S_WorkPos OR
				CO_YPush_Srv_Var.Out_CurrPos <= (H_CO_YPush_Srv_CtnFinalPos - 200) THEN
				CO_YPush_Srv_Var.In_PosCmd := H_CO_YPush_Srv_CurrStandbyPos;
				CO_YPush_Srv_Var.In_VelCmd := A_Srv_YPusherHiSpeed;
				CO_YPush_Srv_Var.In_MoveAbs := TRUE;
				
				CO_FlapGuide_Cyl_Var.In_AutoWork := FALSE;
				CO_FlapGuide_Cyl_Var.In_AutoHome := TRUE;	
			END_IF	

						
			IF 	CO_Brdg_Cyl_Var.S_HomePos AND 
				CO_YPush_Strk_Cyl_Var.S_HomePos AND
				CO_FlapGuide_Cyl_Var.S_HomePos AND
				(CO_YPush_Srv_Var.Out_CurrPos <= (H_CO_YPush_Srv_CtnFinalPos - 600)) 
				AND Station.Run_NextStepPls THEN
			(*	CO_YPush_Srv_Var.In_MoveAbs := FALSE;	*)	
				CO_Brdg_Cyl_Var.In_AutoHome := FALSE;
				CO_FFlapBrdg_Cyl_Var.In_AutoHome := FALSE;
				CO_FlapGuide_Cyl_Var.In_AutoHome := FALSE;
				CO_YPush_Strk_Cyl_Var.In_AutoHome := FALSE;
				
				IF NOT I_CO_YPush_Gap_PE THEN
					Station.SeqFaultWord 	:= 203;	
					E_GapSensor				:= TRUE;	
					Station.SeqFaultString 	:= 'Auto: Bundle Detected at Pusher Gap Sensor Error';												
				ELSE
					Station.RunStep := 200;	(*Flap Closing Can Start After this process*)
				END_IF
			END_IF

			
	200 : 	(************* Wait for Pusher to Reach Home Position  ****************)
			Station.Status 		:= '200: Wait for Pusher to Reach Home Position';
			Station.StatusInt	:= 155;
			CO_YPush_Srv_Var.In_MoveAbs := TRUE;		
			
			IF ((fcComparePos(CurrPos:= CO_YPush_Srv_Var.Out_CurrPos, TargetPos:= CO_YPush_Srv_Var.In_PosCmd, Tolerance := 0.5)) AND
							CO_YPush_Srv_Var.Out_InPos) THEN
				CO_YPush_Srv_Var.In_MoveAbs 	:= FALSE;
				CO_YPush_Cyl_Var.In_AutoWork 	:= FALSE;
				CO_YPush_Cyl_Var.In_AutoHome 	:= TRUE;
				Station.RunStep := 1000;
			END_IF

	1000 : 	(************* Process Done ****************)
			Station.Status 		:= '1000: Process Done';
			Station.StatusInt	:= 499;			
			M_StepRun := FALSE;
			Station.RunStep := 0;
	END_CASE


ELSE
	Station.RunStep := 0;
	
	IF Station.MajorFault OR Station.MinorFault THEN
		Station.Status := 'Station Error';
		Station.StatusInt	:= 4;
	ELSIF Station.Origin THEN
		Station.Status := 'Station In Origin';
		Station.StatusInt	:= 5;
	ELSIF NOT Station.OriginSchRun AND NOT MC.OriginSchRun THEN
		Station.Status := 'Station Not In Origin';
		Station.StatusInt	:= 6;
	END_IF
END_IF

Station.Running := (Station.RunStep>0);

END_PROGRAM

// ---- POUs/MC/Recipe_Handling.TcPOU
PROGRAM Recipe_Handling
VAR
	plsLoadNewRecipe: R_trig;
END_VAR


plsLoadNewRecipe(CLK:=HMI.T_LoadNewRecipe);

IF plsLoadNewRecipe.Q AND NOT MC.AutoMode THEN
	
	(*CurrRecipe := NewRecipe;*)
	
	(* All Gear Ratio to be Set inside Indradrive. Positions are all in mm here*)
	
	H_CO_CV_WA_Srv_TargetPos 		:= 	H_CO_CV_WA_Srv_ZeroOffset - CurrRecipe.rBundleL - 5;
	H_CO_Stopper_WA_Srv_TargetPos 	:= 	H_CO_Stopper_WA_Srv_ZeroOffset - (CurrRecipe.rBundleW * CurrRecipe.iStackX) - 5 ;
	H_CO_FFlapGuide_WA_Srv_TargetPos := H_CO_FFlapGuide_WA_Srv_ZeroOffset -((CurrRecipe.rBundleW + 1) * CurrRecipe.iStackX)  ;
	
	H_ER_FlapL_WA_Srv_TargetPos 	:= H_ER_FlapL_WA_Srv_ZeroOffset - CurrRecipe.rCaseA ;
	H_ER_FlapR_WA_Srv_TargetPos 	:= H_ER_FlapR_WA_Srv_ZeroOffset - CurrRecipe.rCaseA ;	
	
	H_ER_BufCvL_WA_Srv_TargetPos 	:= H_ER_BufCvL_WA_Srv_ZeroOffset -(CurrRecipe.rCaseB/2)-5;
	H_ER_BufCvR_WA_Srv_TargetPos 	:= H_ER_BufCvR_WA_Srv_ZeroOffset -(CurrRecipe.rCaseB/2)-5;
	
	H_ER_WA_Srv_TargetPos 			:= H_ER_WA_Srv_ZeroOffset - CurrRecipe.rCaseC  + 10; (* minus 10mm to over hang the box for 5mm each side*)
	H_EX_HeightL_WA_Srv_TargetPos 	:= H_EX_HeightL_WA_Srv_ZeroOffset - CurrRecipe.rCaseB - 3;
	H_EX_HeightR_WA_Srv_TargetPos 	:= H_EX_HeightR_WA_Srv_ZeroOffset - CurrRecipe.rCaseB - 3;

	
	HMI.T_LoadNewRecipe:=FALSE;
	
END_IF

END_PROGRAM

// ---- POUs/MC/Emergency_Stop.TcPOU
PROGRAM Emergency_Stop
VAR
	EmergencyStop_Fault	: BOOL;	
	tmrEmergencyStop	: Ton;
END_VAR


EmergencyStop_Fault	:= 	E_Estop_Panel		OR
						E_Estop_Collator	OR
						E_Estop_HorLeft		OR
						E_Estop_HorRight 	OR
						E_Estop_HorExit ;

tmrEmergencyStop (IN := (EmergencyStop_Fault AND I_Emg_SC_OK ) OR (NOT EmergencyStop_Fault AND not I_Emg_SC_OK ), pt:= T#1S);
(*
IF tmrEmergencyStop.Q THEN
E_EStop_SafetyBroken	:= TRUE;						
END_IF															
*)						
IF mc.ResetPressed THEN
	E_Estop_Panel			:= FALSE;
	E_Estop_Collator		:= FALSE;
	E_Estop_HorLeft			:= FALSE;
	E_Estop_HorRight		:= FALSE;
	E_Estop_HorExit			:= FALSE;
	E_EStop_SafetyBroken	:= FALSE;
END_IF

(*
IF NOT I_EStop_Panel THEN
	E_Estop_Panel		:= TRUE;
END_IF

IF NOT I_EStop_Collator THEN
	E_Estop_Collator	:= TRUE;
END_IF

IF NOT I_EStop_HorL THEN
	E_Estop_HorLeft		:= TRUE;
END_IF

IF NOT I_EStop_HorR THEN
	E_Estop_HorRight	:= TRUE;
END_IF

IF NOT I_EStop_HorExit THEN
	E_Estop_HorExit		:= TRUE;
END_IF
*)

END_PROGRAM

// ---- POUs/Collator/CO_Main.TcPOU
PROGRAM CO_Main
VAR
	i: INT;
END_VAR

IF Cfg_BypassCollator THEN
	HMI.T_Station_BypassP[0] := TRUE;
	HMI.T_Station_BypassP[1] := TRUE;
	HMI.T_Station_BypassP[2] := TRUE;
ELSE
	HMI.T_Station_BypassP[0] := FALSE;
	HMI.T_Station_BypassP[1] := FALSE;
	HMI.T_Station_BypassP[2] := FALSE;
END_IF

I_CO_YPush_Gap_PE := TRUE;	(*Simulate Gap Sensor, No Hardware sensor*)

CO_Timers();
(* Previously known as stacker *)
sc[0].Origin	:= TRUE;
sc[0].Name		:= 'Spare Station';

(* Previously known as XPusher *)
sc[1].Origin	:= TRUE;
sc[1].Name		:= 'Spare Station';

CO_YPush_Error	(Station:= SC[2]);
CO_YPush_Auto	(Station:= SC[2]);
CO_YPush_Origin	(Station:= SC[2]);
SC[2].T_OriginSearch := CO_YPush.T_OriginSearch;
CO_YPush := SC[2];

CO_Cylinder_Output();
CO_Servo_Output();
CO_Nordson();

(* CO Structure is only for displaying on HMI*)
CO.Origin := SC[0].Origin AND SC[1].Origin AND SC[2].Origin;
CO.MajorFault := SC[0].MajorFault OR SC[1].MajorFault OR SC[2].MajorFault;
CO.MinorFault := SC[0].MinorFault OR SC[1].MinorFault OR SC[2].MinorFault;
CO.Warning := SC[0].Warning OR SC[1].Warning OR SC[2].Warning;
CO.AutoRun := SC[0].AutoRun OR SC[1].AutoRun OR SC[2].AutoRun;
CO.Running := SC[0].Running OR SC[1].Running OR SC[2].Running;
CO.OriginSchRun := SC[0].OriginSchRun OR SC[1].OriginSchRun OR SC[2].OriginSchRun;

END_PROGRAM

// ---- POUs/Collator/CO_Timers.TcPOU
PROGRAM CO_Timers
VAR
END_VAR


CO_Stk_Up_TON (IN := I_CO_Stk_Mtr_UpPos, pt := T#0MS);

CO_Stk_Dn_TON (IN := I_CO_Stk_Mtr_HomePos, pt := T#30MS);

CO_Bdl_Reach_TON (IN := I_CO_Bdl_PE1, pt := T#100MS);	(*End of Stacking Conveyor*)

CO_Bdl_Stack_TON (IN := I_CO_Bdl_Stack_PE, pt := T#100MS);

CO_Stk_AtBuf_TON (IN := I_CO_YStk_AtBuf1_PE, pt := T#100MS);

CO_Bdl_ZFull_TON (IN := I_CO_Bdl_ZFull_PE AND NOT I_CO_Bdl_ZLimit_PE, pt := T#1S);

CO_Bdl_ZFull_TOFF (IN := NOT I_CO_Bdl_ZFull_PE AND NOT I_CO_Bdl_ZLimit_PE, pt := T#1S);

END_PROGRAM

// ---- POUs/Collator/Y Pusher n Bridge/CO_YPush_Error.TcPOU
PROGRAM CO_YPush_Error
VAR_IN_OUT
	Station		:structStationCtrl;
END_VAR

VAR
END_VAR

IF MC.ResetPressed THEN
	Station.SeqFaultWord := 0;
END_IF

(* 	Reserved Station.SeqFaultWord 
	= 1~49 for Major Fault
	= 100~149 for Origin Sequence Fault
	= 150~199 for Origin Width Adjust Sequence Fault
	= 200~299 for Auto Sequence Fault
	= 300~399 for misc fault listed on this page*)

Station.MajorFault := (Station.SeqFaultWord > 0) AND (Station.SeqFaultWord < 50);
Station.MinorFault := (Station.SeqFaultWord >= 100) OR Station.DeviceFault or E_PTC_BundleNOK;

END_PROGRAM

// ---- POUs/Collator/Y Pusher n Bridge/CO_YPush_Origin.TcPOU
PROGRAM CO_YPush_Origin
VAR_IN_OUT
	Station		:structStationCtrl;
END_VAR
VAR
	CO_YPush_WA_Origin: BOOL;
	pls_OriginSchRun: R_trig;
END_VAR

(**************************************************************************************************************)
(* Station Width Adjust in Origin Condition *)
(**************************************************************************************************************)
CO_YPush_WA_Origin := TRUE;

(**************************************************************************************************************)
(* Station Origin Condition *)
(**************************************************************************************************************)

H_CO_YPush_Srv_CurrStandbyPos := H_CO_YPush_Srv_HomePos;
					(*offset 200.0 because box size of 200 is used during teaching*)

Station.Origin 	:=	(CO_YPush_WA_Origin 			AND 
					CO_YPush_Strk_Cyl_Var.S_HomePos AND
					CO_YPush_Cyl_Var.S_HomePos 		AND
					(((fcComparePos(CurrPos:= CO_YPush_Srv_Var.Out_CurrPos, TargetPos:= H_CO_YPush_Srv_CurrStandbyPos, Tolerance := 0.5)) AND
							CO_YPush_Srv_Var.Out_InPos AND CO_YPush_Srv_Var.Out_Ready)) AND
					CO_Brdg_Cyl_Var.S_HomePos AND 
					CO_FlapGuide_Cyl_Var.S_HomePos) OR
					Station.Bypass
					;
					 		
(**************************************************************************************************************)
(* Station Origin Step *)
(**************************************************************************************************************)

pls_OriginSchRun(CLK:= (MC.OriginSchRun OR Station.OriginSchRun) );

IF (MC.OriginSchRun OR Station.OriginSchRun) AND NOT Station.Bypass   THEN
	CASE Station.OriginRunStep OF

	0 : 	(************* Ready To Run ****************)
			IF NOT Station.Origin AND pls_OriginSchRun.Q THEN
				Station.OriginRunStep := Station.OriginRunStep+10;	
			END_IF

